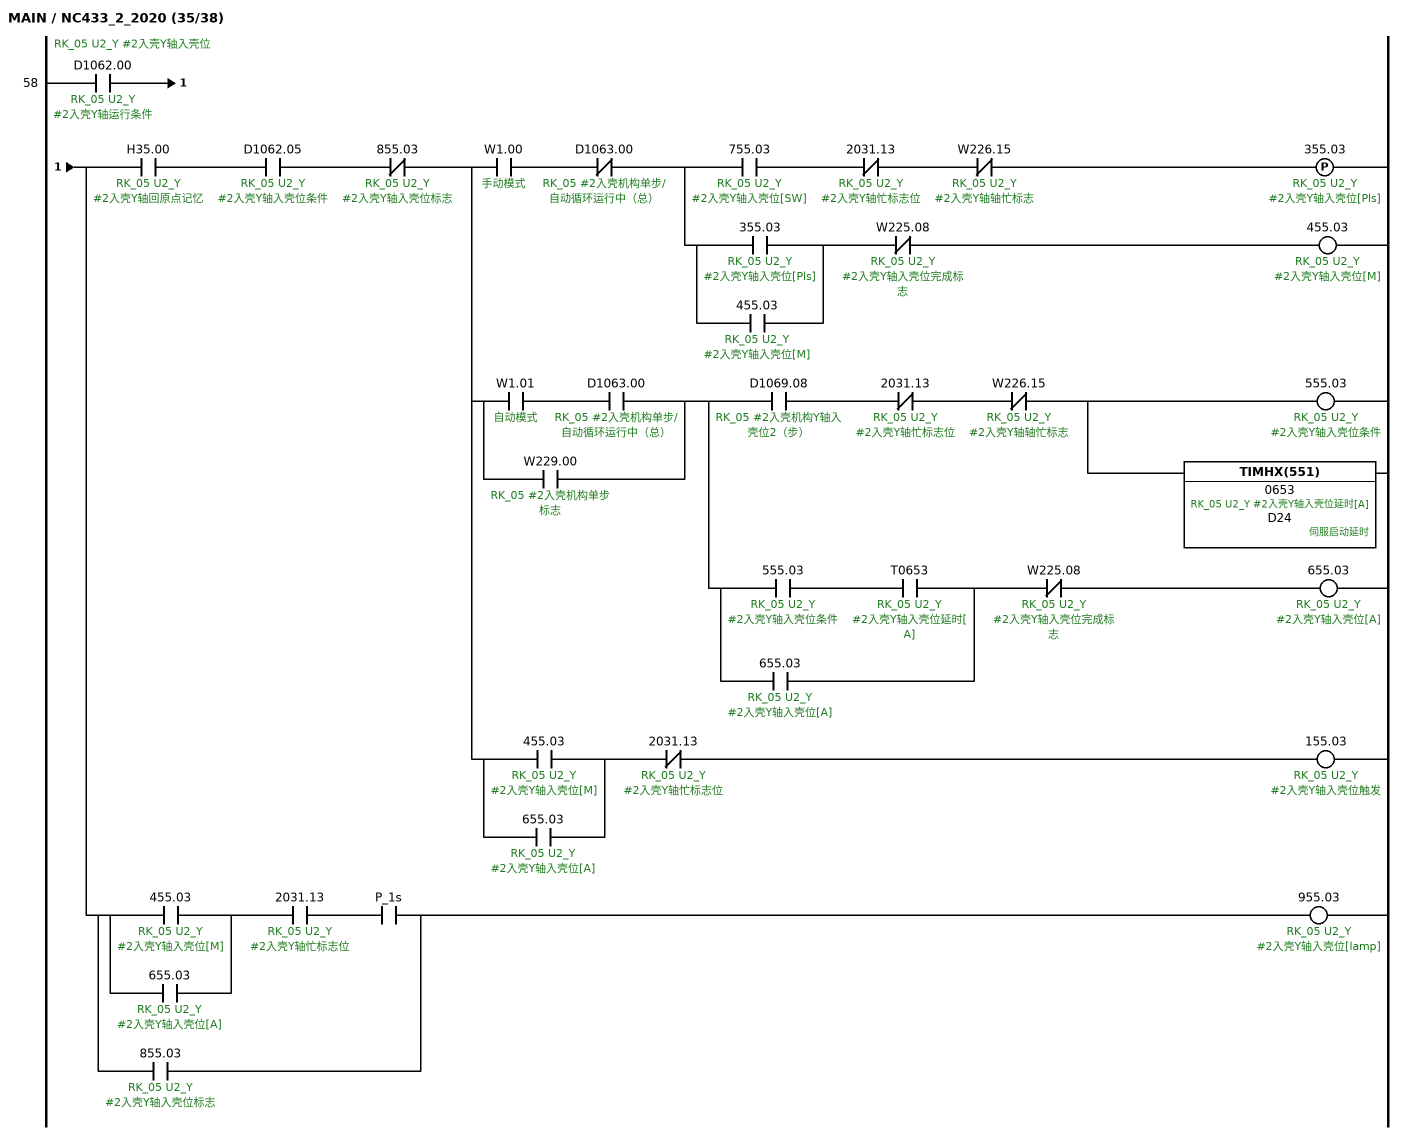
; [picture p144: MAIN / NC433_2_2020, rungs 58-58]
; rung 58: RK_05 U2_Y #2入壳Y轴入壳位
LD D1062.00  ; RK_05 U2_Y #2入壳Y轴运行条件
OUT TR0
AND H35.00  ; RK_05 U2_Y #2入壳Y轴回原点记忆
AND D1062.05  ; RK_05 U2_Y #2入壳Y轴入壳位条件
ANDNOT 855.03  ; RK_05 U2_Y #2入壳Y轴入壳位标志
OUT TR1
AND W1.00  ; 手动模式
ANDNOT D1063.00  ; RK_05 #2入壳机构单步/自动循环运行中（总）
OUT TR2
AND 755.03  ; RK_05 U2_Y #2入壳Y轴入壳位[SW]
ANDNOT 2031.13  ; RK_05 U2_Y #2入壳Y轴忙标志位
ANDNOT W226.15  ; RK_05 U2_Y #2入壳Y轴轴忙标志
DIFU(013) 355.03  ; RK_05 U2_Y #2入壳Y轴入壳位[Pls]
LD TR2
LD 355.03  ; RK_05 U2_Y #2入壳Y轴入壳位[Pls]
OR 455.03  ; RK_05 U2_Y #2入壳Y轴入壳位[M]
ANDLD
ANDNOT W225.08  ; RK_05 U2_Y #2入壳Y轴入壳位完成标志
OUT 455.03  ; RK_05 U2_Y #2入壳Y轴入壳位[M]
LD TR1
LD W1.01  ; 自动模式
AND D1063.00  ; RK_05 #2入壳机构单步/自动循环运行中（总）
OR W229.00  ; RK_05 #2入壳机构单步标志
ANDLD
OUT TR2
AND D1069.08  ; RK_05 #2入壳机构Y轴入壳位2（步）
ANDNOT 2031.13  ; RK_05 U2_Y #2入壳Y轴忙标志位
ANDNOT W226.15  ; RK_05 U2_Y #2入壳Y轴轴忙标志
OUT 555.03  ; RK_05 U2_Y #2入壳Y轴入壳位条件
TIMHX(551) 0653 D24  ; 伺服启动延时, RK_05 U2_Y #2入壳Y轴入壳位延时[A]
LD TR2
LD 555.03  ; RK_05 U2_Y #2入壳Y轴入壳位条件
AND T0653  ; RK_05 U2_Y #2入壳Y轴入壳位延时[A]
OR 655.03  ; RK_05 U2_Y #2入壳Y轴入壳位[A]
ANDLD
ANDNOT W225.08  ; RK_05 U2_Y #2入壳Y轴入壳位完成标志
OUT 655.03  ; RK_05 U2_Y #2入壳Y轴入壳位[A]
LD TR1
LD 455.03  ; RK_05 U2_Y #2入壳Y轴入壳位[M]
OR 655.03  ; RK_05 U2_Y #2入壳Y轴入壳位[A]
ANDLD
ANDNOT 2031.13  ; RK_05 U2_Y #2入壳Y轴忙标志位
OUT 155.03  ; RK_05 U2_Y #2入壳Y轴入壳位触发
LD TR0
LD 455.03  ; RK_05 U2_Y #2入壳Y轴入壳位[M]
OR 655.03  ; RK_05 U2_Y #2入壳Y轴入壳位[A]
AND 2031.13  ; RK_05 U2_Y #2入壳Y轴忙标志位
AND P_1s
OR 855.03  ; RK_05 U2_Y #2入壳Y轴入壳位标志
ANDLD
OUT 955.03  ; RK_05 U2_Y #2入壳Y轴入壳位[lamp]

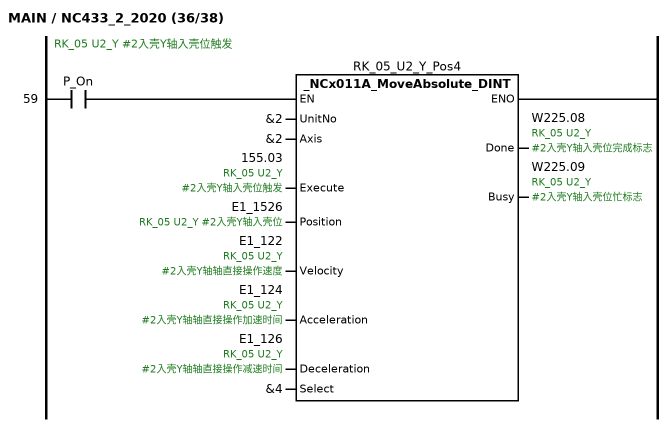
; rung 59: RK_05 U2_Y #2入壳Y轴入壳位触发
LD P_On
CALL RK_05_U2_Y_Pos4 : _NCx011A_MoveAbsolute_DINT (UnitNo := &2, Axis := &2, Execute := 155.03, Position := E1_1526, Velocity := E1_122, Acceleration := E1_124, Deceleration := E1_126, Select := &4, Done => W225.08, Busy => W225.09)  ; RK_05 U2_Y #2入壳Y轴入壳位触发, RK_05 U2_Y #2入壳Y轴入壳位, RK_05 U2_Y #2入壳Y轴轴直接操作速度, RK_05 U2_Y #2入壳Y轴轴直接操作加速时间, RK_05 U2_Y #2入壳Y轴轴直接操作减速时间, RK_05 U2_Y #2入壳Y轴入壳位完成标志, RK_05 U2_Y #2入壳Y轴入壳位忙标志

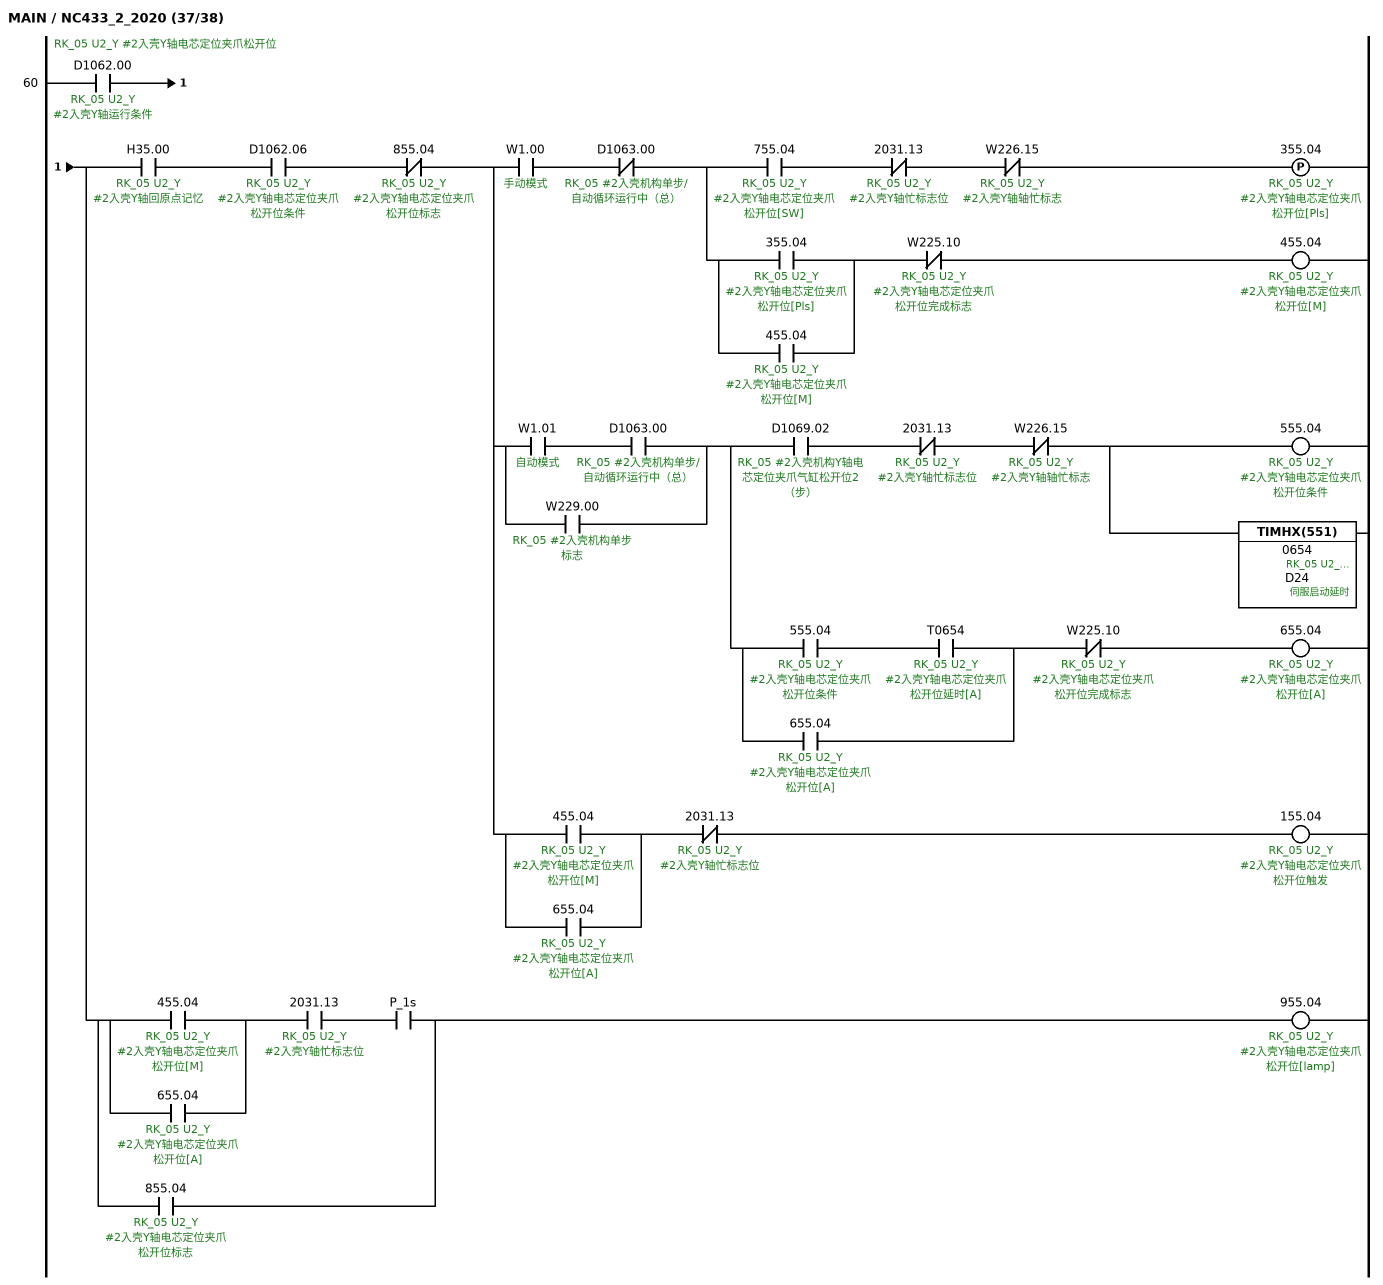
; rung 60: RK_05 U2_Y #2入壳Y轴电芯定位夹爪松开位
LD D1062.00  ; RK_05 U2_Y #2入壳Y轴运行条件
OUT TR0
AND H35.00  ; RK_05 U2_Y #2入壳Y轴回原点记忆
AND D1062.06  ; RK_05 U2_Y #2入壳Y轴电芯定位夹爪松开位条件
ANDNOT 855.04  ; RK_05 U2_Y #2入壳Y轴电芯定位夹爪松开位标志
OUT TR1
AND W1.00  ; 手动模式
ANDNOT D1063.00  ; RK_05 #2入壳机构单步/自动循环运行中（总）
OUT TR2
AND 755.04  ; RK_05 U2_Y #2入壳Y轴电芯定位夹爪松开位[SW]
ANDNOT 2031.13  ; RK_05 U2_Y #2入壳Y轴忙标志位
ANDNOT W226.15  ; RK_05 U2_Y #2入壳Y轴轴忙标志
DIFU(013) 355.04  ; RK_05 U2_Y #2入壳Y轴电芯定位夹爪松开位[Pls]
LD TR2
LD 355.04  ; RK_05 U2_Y #2入壳Y轴电芯定位夹爪松开位[Pls]
OR 455.04  ; RK_05 U2_Y #2入壳Y轴电芯定位夹爪松开位[M]
ANDLD
ANDNOT W225.10  ; RK_05 U2_Y #2入壳Y轴电芯定位夹爪松开位完成标志
OUT 455.04  ; RK_05 U2_Y #2入壳Y轴电芯定位夹爪松开位[M]
LD TR1
LD W1.01  ; 自动模式
AND D1063.00  ; RK_05 #2入壳机构单步/自动循环运行中（总）
OR W229.00  ; RK_05 #2入壳机构单步标志
ANDLD
OUT TR2
AND D1069.02  ; RK_05 #2入壳机构Y轴电芯定位夹爪气缸松开位2（步）
ANDNOT 2031.13  ; RK_05 U2_Y #2入壳Y轴忙标志位
ANDNOT W226.15  ; RK_05 U2_Y #2入壳Y轴轴忙标志
OUT 555.04  ; RK_05 U2_Y #2入壳Y轴电芯定位夹爪松开位条件
TIMHX(551) 0654 D24  ; 伺服启动延时, RK_05 U2_Y #2入壳Y轴电芯定位夹爪松开位延时[A]
LD TR2
LD 555.04  ; RK_05 U2_Y #2入壳Y轴电芯定位夹爪松开位条件
AND T0654  ; RK_05 U2_Y #2入壳Y轴电芯定位夹爪松开位延时[A]
OR 655.04  ; RK_05 U2_Y #2入壳Y轴电芯定位夹爪松开位[A]
ANDLD
ANDNOT W225.10  ; RK_05 U2_Y #2入壳Y轴电芯定位夹爪松开位完成标志
OUT 655.04  ; RK_05 U2_Y #2入壳Y轴电芯定位夹爪松开位[A]
LD TR1
LD 455.04  ; RK_05 U2_Y #2入壳Y轴电芯定位夹爪松开位[M]
OR 655.04  ; RK_05 U2_Y #2入壳Y轴电芯定位夹爪松开位[A]
ANDLD
ANDNOT 2031.13  ; RK_05 U2_Y #2入壳Y轴忙标志位
OUT 155.04  ; RK_05 U2_Y #2入壳Y轴电芯定位夹爪松开位触发
LD TR0
LD 455.04  ; RK_05 U2_Y #2入壳Y轴电芯定位夹爪松开位[M]
OR 655.04  ; RK_05 U2_Y #2入壳Y轴电芯定位夹爪松开位[A]
AND 2031.13  ; RK_05 U2_Y #2入壳Y轴忙标志位
AND P_1s
OR 855.04  ; RK_05 U2_Y #2入壳Y轴电芯定位夹爪松开位标志
ANDLD
OUT 955.04  ; RK_05 U2_Y #2入壳Y轴电芯定位夹爪松开位[lamp]

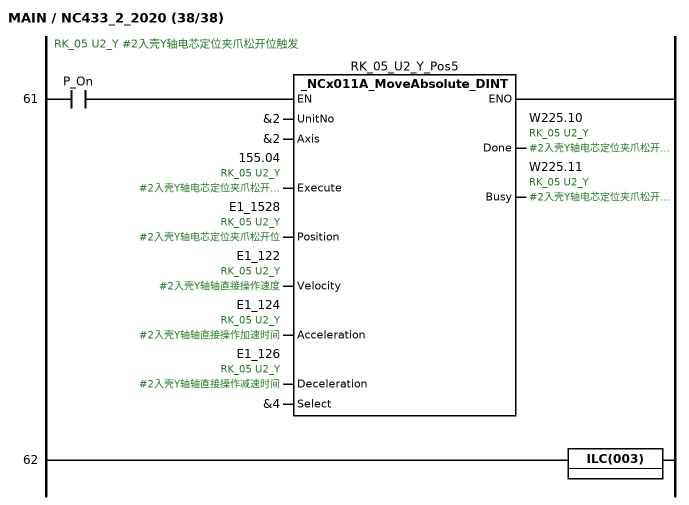
; rung 61: RK_05 U2_Y #2入壳Y轴电芯定位夹爪松开位触发
LD P_On
CALL RK_05_U2_Y_Pos5 : _NCx011A_MoveAbsolute_DINT (UnitNo := &2, Axis := &2, Execute := 155.04, Position := E1_1528, Velocity := E1_122, Acceleration := E1_124, Deceleration := E1_126, Select := &4, Done => W225.10, Busy => W225.11)  ; RK_05 U2_Y #2入壳Y轴电芯定位夹爪松开位触发, RK_05 U2_Y #2入壳Y轴电芯定位夹爪松开位, RK_05 U2_Y #2入壳Y轴轴直接操作速度, RK_05 U2_Y #2入壳Y轴轴直接操作加速时间, RK_05 U2_Y #2入壳Y轴轴直接操作减速时间, RK_05 U2_Y #2入壳Y轴电芯定位夹爪松开位完成标志, RK_05 U2_Y #2入壳Y轴电芯定位夹爪松开位忙标志
; rung 62
ILC(003)

### Section NC433_4_2040

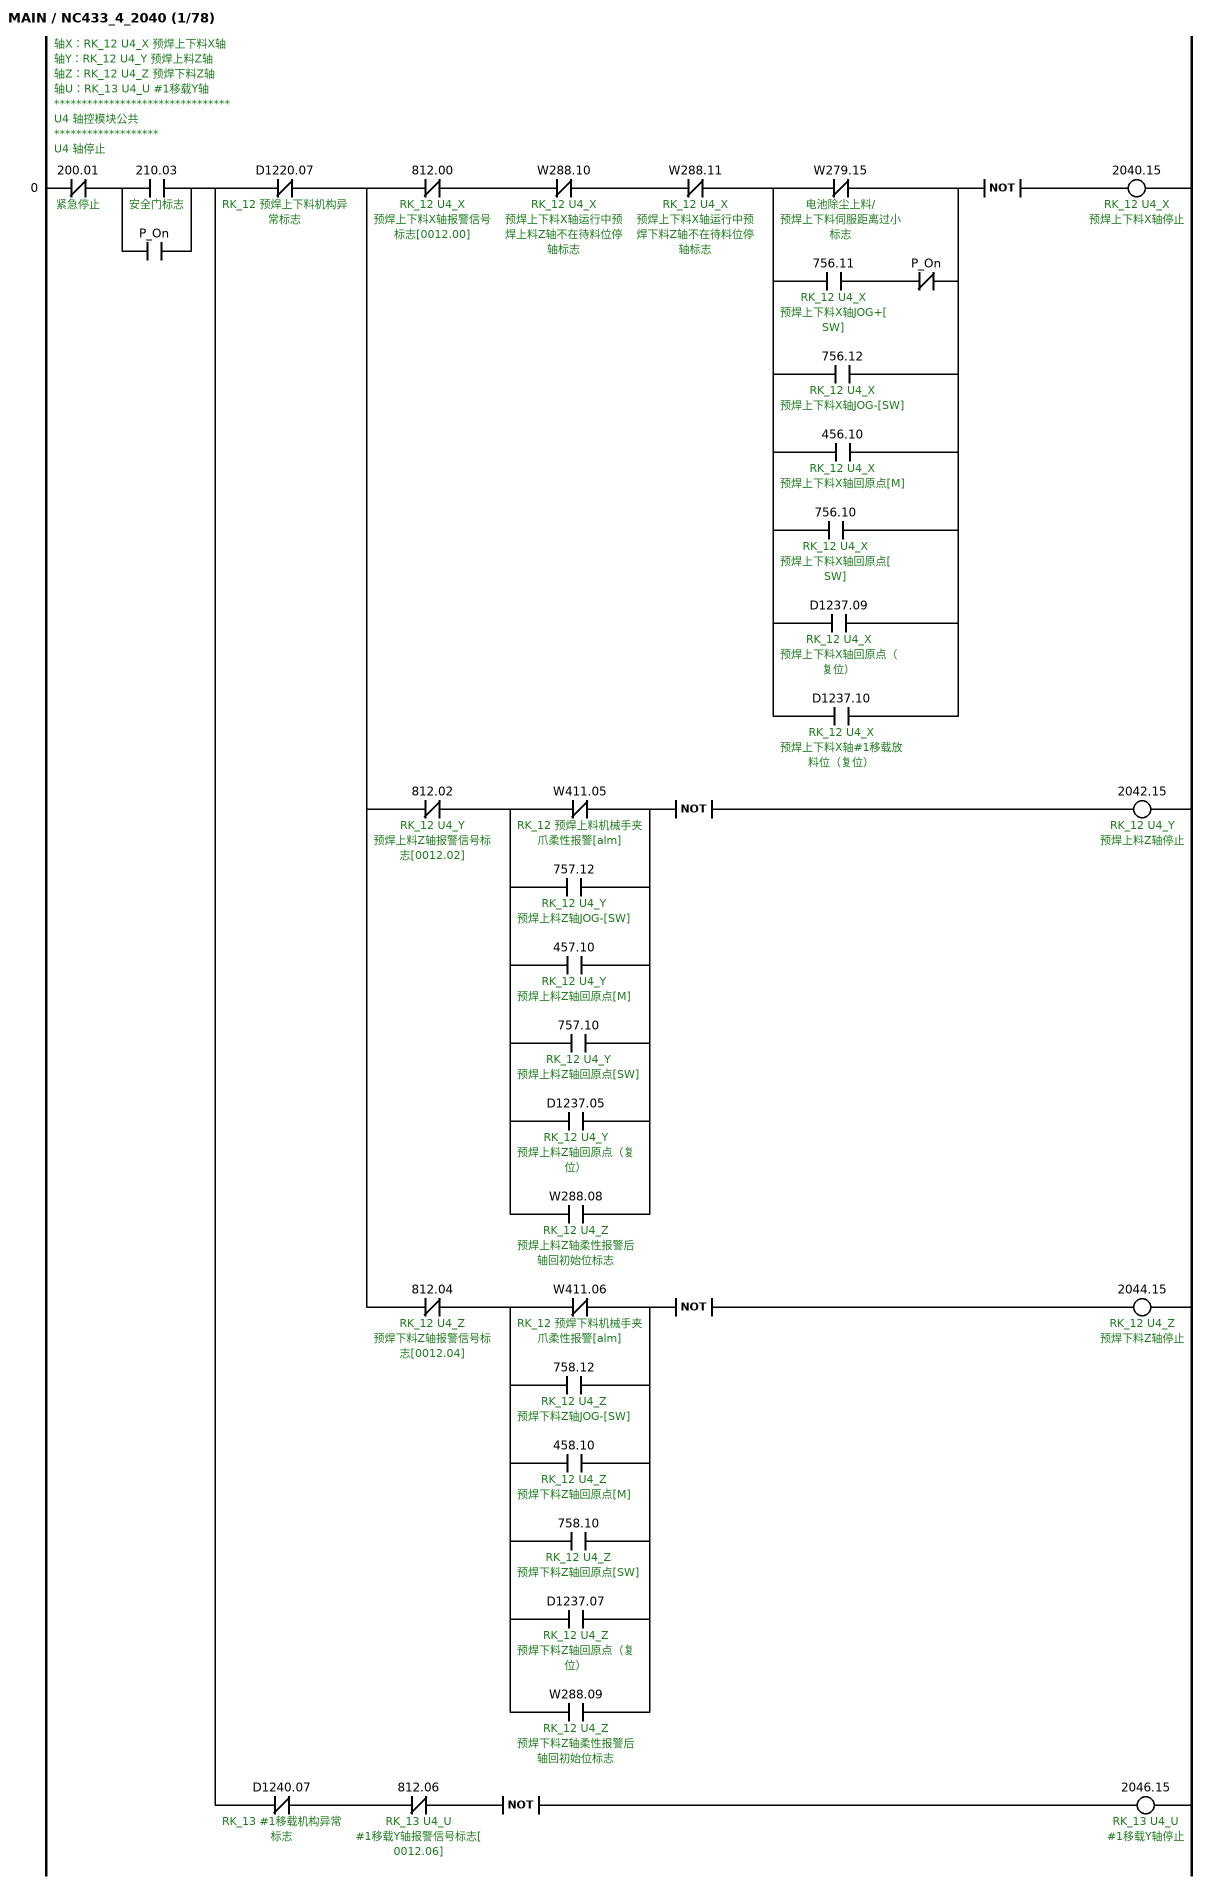
; rung 0: 轴X：RK_12 U4_X 预焊上下料X轴 / 轴Y：RK_12 U4_Y 预焊上料Z轴 / 轴Z：RK_12 U4_Z 预焊下料Z轴 / 轴U：RK_13 U4_U #1移载Y轴 / ******************************** / U4 轴控模块公共 / ******************* / U4 轴停止
LDNOT 200.01  ; 紧急停止
LD 210.03  ; 安全门标志
OR P_On
ANDLD
OUT TR0
ANDNOT D1220.07  ; RK_12 预焊上下料机构异常标志
OUT TR1
ANDNOT 812.00  ; RK_12 U4_X 预焊上下料X轴报警信号标志[0012.00]
ANDNOT W288.10  ; RK_12 U4_X 预焊上下料X轴运行中预焊上料Z轴不在待料位停轴标志
ANDNOT W288.11  ; RK_12 U4_X 预焊上下料X轴运行中预焊下料Z轴不在待料位停轴标志
LDNOT W279.15  ; 电池除尘上料/预焊上下料伺服距离过小标志
LD 756.11  ; RK_12 U4_X 预焊上下料X轴JOG+[SW]
ANDNOT P_On
ORLD
OR 756.12  ; RK_12 U4_X 预焊上下料X轴JOG-[SW]
OR 456.10  ; RK_12 U4_X 预焊上下料X轴回原点[M]
OR 756.10  ; RK_12 U4_X 预焊上下料X轴回原点[SW]
OR D1237.09  ; RK_12 U4_X 预焊上下料X轴回原点（复位）
OR D1237.10  ; RK_12 U4_X 预焊上下料X轴#1移载放料位（复位）
ANDLD
NOT(520)
OUT 2040.15  ; RK_12 U4_X 预焊上下料X轴停止
LD TR1
ANDNOT 812.02  ; RK_12 U4_Y 预焊上料Z轴报警信号标志[0012.02]
LDNOT W411.05  ; RK_12 预焊上料机械手夹爪柔性报警[alm]
OR 757.12  ; RK_12 U4_Y 预焊上料Z轴JOG-[SW]
OR 457.10  ; RK_12 U4_Y 预焊上料Z轴回原点[M]
OR 757.10  ; RK_12 U4_Y 预焊上料Z轴回原点[SW]
OR D1237.05  ; RK_12 U4_Y 预焊上料Z轴回原点（复位）
OR W288.08  ; RK_12 U4_Z 预焊上料Z轴柔性报警后轴回初始位标志
ANDLD
NOT(520)
OUT 2042.15  ; RK_12 U4_Y 预焊上料Z轴停止
LD TR1
ANDNOT 812.04  ; RK_12 U4_Z 预焊下料Z轴报警信号标志[0012.04]
LDNOT W411.06  ; RK_12 预焊下料机械手夹爪柔性报警[alm]
OR 758.12  ; RK_12 U4_Z 预焊下料Z轴JOG-[SW]
OR 458.10  ; RK_12 U4_Z 预焊下料Z轴回原点[M]
OR 758.10  ; RK_12 U4_Z 预焊下料Z轴回原点[SW]
OR D1237.07  ; RK_12 U4_Z 预焊下料Z轴回原点（复位）
OR W288.09  ; RK_12 U4_Z 预焊下料Z轴柔性报警后轴回初始位标志
ANDLD
NOT(520)
OUT 2044.15  ; RK_12 U4_Z 预焊下料Z轴停止
LD TR0
ANDNOT D1240.07  ; RK_13 #1移载机构异常标志
ANDNOT 812.06  ; RK_13 U4_U #1移载Y轴报警信号标志[0012.06]
NOT(520)
OUT 2046.15  ; RK_13 U4_U #1移载Y轴停止

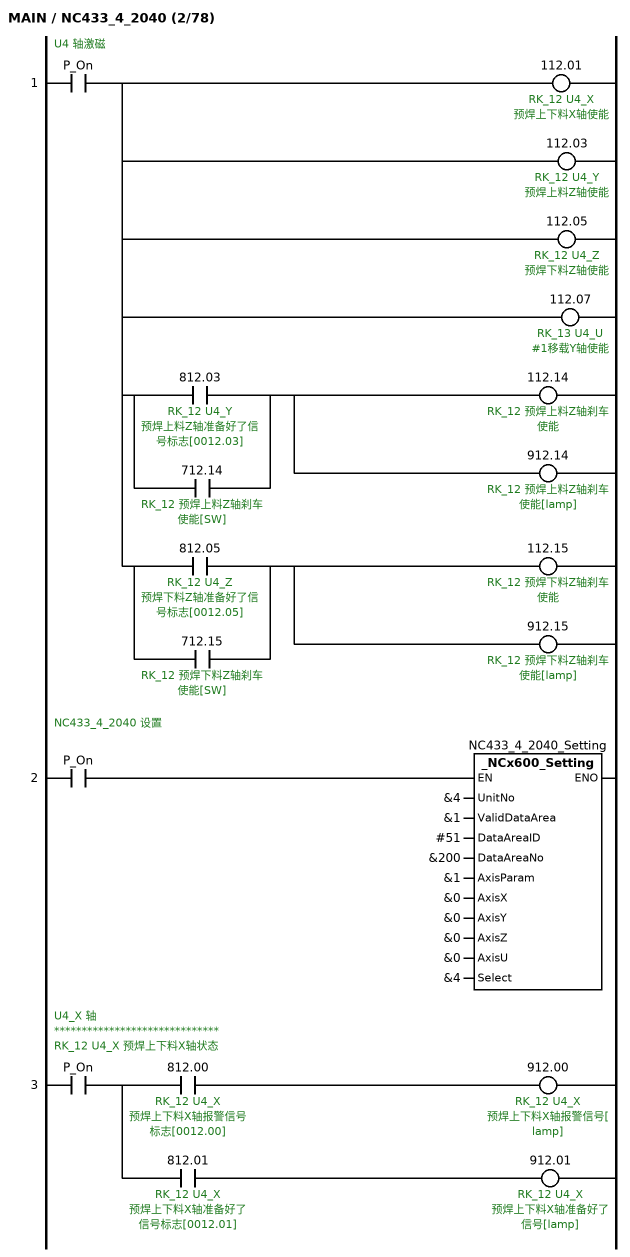
; rung 1: U4 轴激磁
LD P_On
OUT TR0
OUT 112.01  ; RK_12 U4_X 预焊上下料X轴使能
OUT 112.03  ; RK_12 U4_Y 预焊上料Z轴使能
OUT 112.05  ; RK_12 U4_Z 预焊下料Z轴使能
OUT 112.07  ; RK_13 U4_U #1移载Y轴使能
LD 812.03  ; RK_12 U4_Y 预焊上料Z轴准备好了信号标志[0012.03]
OR 712.14  ; RK_12 预焊上料Z轴刹车使能[SW]
ANDLD
OUT 112.14  ; RK_12 预焊上料Z轴刹车使能
OUT 912.14  ; RK_12 预焊上料Z轴刹车使能[lamp]
LD TR0
LD 812.05  ; RK_12 U4_Z 预焊下料Z轴准备好了信号标志[0012.05]
OR 712.15  ; RK_12 预焊下料Z轴刹车使能[SW]
ANDLD
OUT 112.15  ; RK_12 预焊下料Z轴刹车使能
OUT 912.15  ; RK_12 预焊下料Z轴刹车使能[lamp]
; rung 2: NC433_4_2040 设置
LD P_On
CALL NC433_4_2040_Setting : _NCx600_Setting (UnitNo := &4, ValidDataArea := &1, DataAreaID := #51, DataAreaNo := &200, AxisParam := &1, AxisX := &0, AxisY := &0, AxisZ := &0, AxisU := &0, Select := &4)
; rung 3: U4_X 轴 / ****************************** / RK_12 U4_X 预焊上下料X轴状态
LD P_On
OUT TR0
AND 812.00  ; RK_12 U4_X 预焊上下料X轴报警信号标志[0012.00]
OUT 912.00  ; RK_12 U4_X 预焊上下料X轴报警信号[lamp]
LD TR0
AND 812.01  ; RK_12 U4_X 预焊上下料X轴准备好了信号标志[0012.01]
OUT 912.01  ; RK_12 U4_X 预焊上下料X轴准备好了信号[lamp]

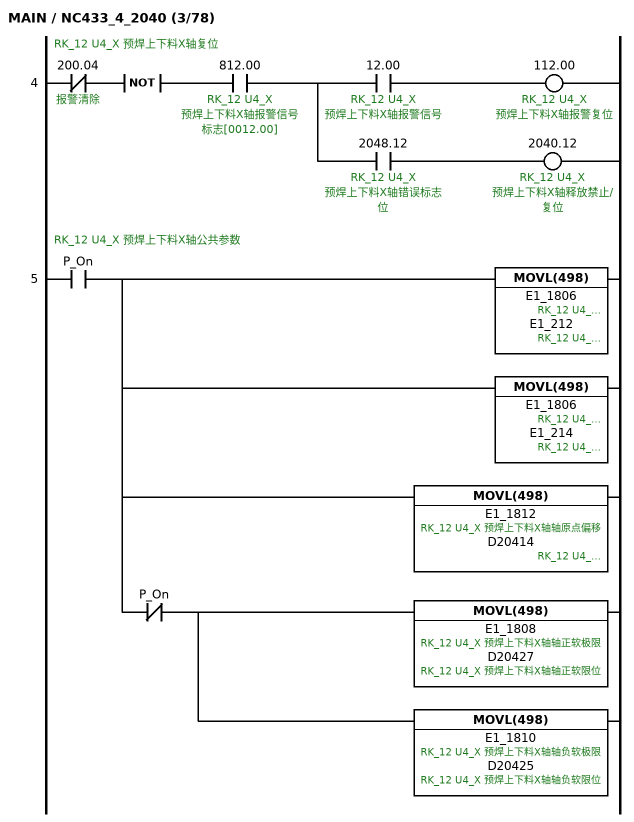
; rung 4: RK_12 U4_X 预焊上下料X轴复位
LDNOT 200.04  ; 报警清除
NOT(520)
AND 812.00  ; RK_12 U4_X 预焊上下料X轴报警信号标志[0012.00]
OUT TR0
AND 12.00  ; RK_12 U4_X 预焊上下料X轴报警信号
OUT 112.00  ; RK_12 U4_X 预焊上下料X轴报警复位
LD TR0
AND 2048.12  ; RK_12 U4_X 预焊上下料X轴错误标志位
OUT 2040.12  ; RK_12 U4_X 预焊上下料X轴释放禁止/复位
; rung 5: RK_12 U4_X 预焊上下料X轴公共参数
LD P_On
MOVL(498) E1_1806 E1_212  ; RK_12 U4_X 预焊上下料X轴轴加减速时间, RK_12 U4_X 预焊上下料X轴轴直接操作加速时间
MOVL(498) E1_1806 E1_214  ; RK_12 U4_X 预焊上下料X轴轴加减速时间, RK_12 U4_X 预焊上下料X轴轴直接操作减速时间
MOVL(498) E1_1812 D20414  ; RK_12 U4_X 预焊上下料X轴轴原点偏移, RK_12 U4_X 预焊上下料X轴轴原点补偿值
ANDNOT P_On
MOVL(498) E1_1808 D20427  ; RK_12 U4_X 预焊上下料X轴轴正软极限, RK_12 U4_X 预焊上下料X轴轴正软限位
MOVL(498) E1_1810 D20425  ; RK_12 U4_X 预焊上下料X轴轴负软极限, RK_12 U4_X 预焊上下料X轴轴负软限位

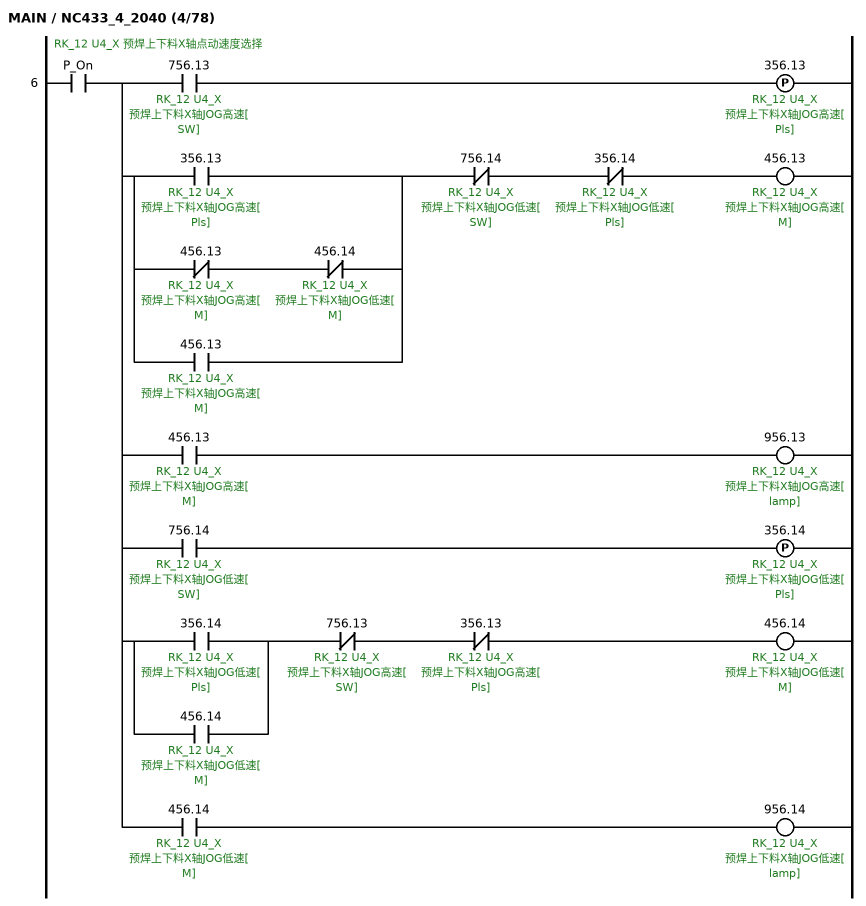
; rung 6: RK_12 U4_X 预焊上下料X轴点动速度选择
LD P_On
OUT TR0
AND 756.13  ; RK_12 U4_X 预焊上下料X轴JOG高速[SW]
DIFU(013) 356.13  ; RK_12 U4_X 预焊上下料X轴JOG高速[Pls]
LD TR0
LD 356.13  ; RK_12 U4_X 预焊上下料X轴JOG高速[Pls]
LDNOT 456.13  ; RK_12 U4_X 预焊上下料X轴JOG高速[M]
ANDNOT 456.14  ; RK_12 U4_X 预焊上下料X轴JOG低速[M]
ORLD
OR 456.13  ; RK_12 U4_X 预焊上下料X轴JOG高速[M]
ANDLD
ANDNOT 756.14  ; RK_12 U4_X 预焊上下料X轴JOG低速[SW]
ANDNOT 356.14  ; RK_12 U4_X 预焊上下料X轴JOG低速[Pls]
OUT 456.13  ; RK_12 U4_X 预焊上下料X轴JOG高速[M]
LD TR0
AND 456.13  ; RK_12 U4_X 预焊上下料X轴JOG高速[M]
OUT 956.13  ; RK_12 U4_X 预焊上下料X轴JOG高速[lamp]
LD TR0
AND 756.14  ; RK_12 U4_X 预焊上下料X轴JOG低速[SW]
DIFU(013) 356.14  ; RK_12 U4_X 预焊上下料X轴JOG低速[Pls]
LD TR0
LD 356.14  ; RK_12 U4_X 预焊上下料X轴JOG低速[Pls]
OR 456.14  ; RK_12 U4_X 预焊上下料X轴JOG低速[M]
ANDLD
ANDNOT 756.13  ; RK_12 U4_X 预焊上下料X轴JOG高速[SW]
ANDNOT 356.13  ; RK_12 U4_X 预焊上下料X轴JOG高速[Pls]
OUT 456.14  ; RK_12 U4_X 预焊上下料X轴JOG低速[M]
LD TR0
AND 456.14  ; RK_12 U4_X 预焊上下料X轴JOG低速[M]
OUT 956.14  ; RK_12 U4_X 预焊上下料X轴JOG低速[lamp]

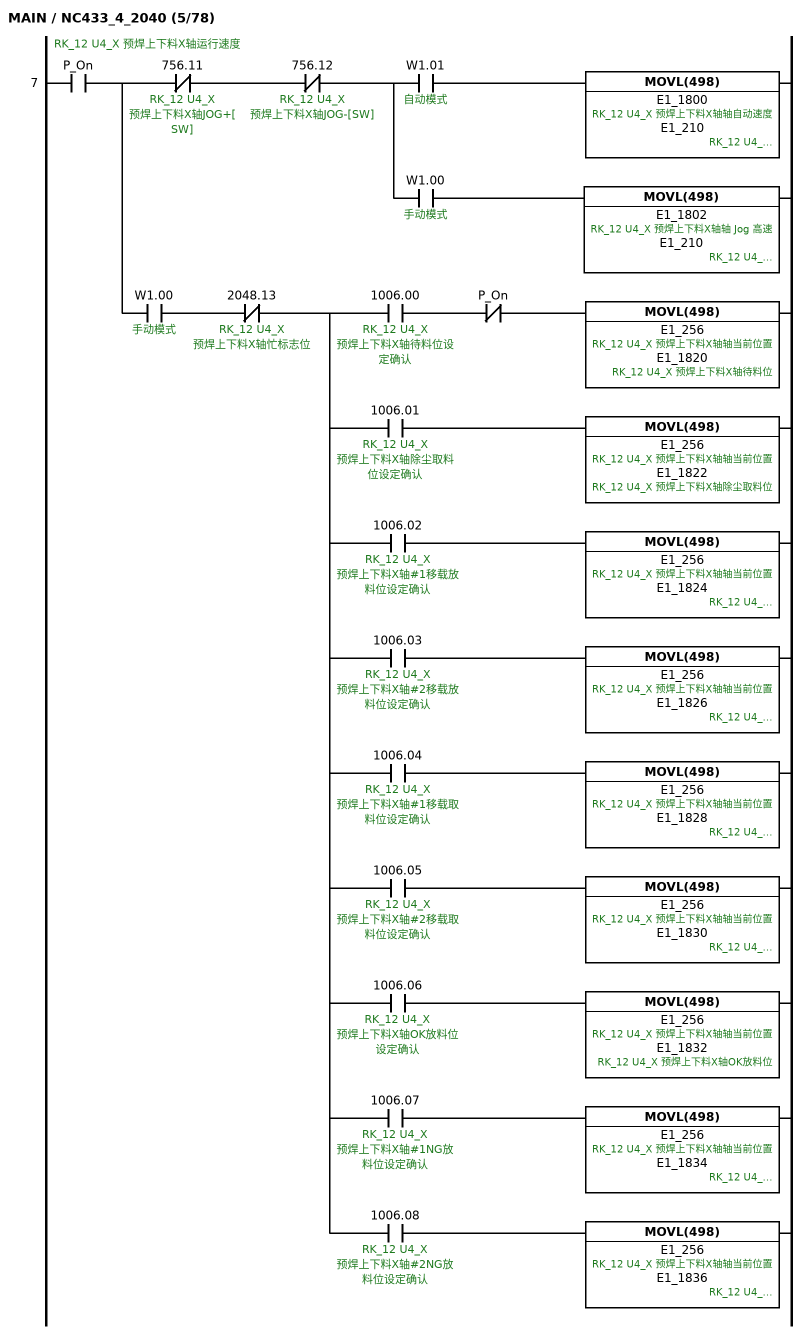
; rung 7: RK_12 U4_X 预焊上下料X轴运行速度
LD P_On
OUT TR0
ANDNOT 756.11  ; RK_12 U4_X 预焊上下料X轴JOG+[SW]
ANDNOT 756.12  ; RK_12 U4_X 预焊上下料X轴JOG-[SW]
OUT TR1
AND W1.01  ; 自动模式
MOVL(498) E1_1800 E1_210  ; RK_12 U4_X 预焊上下料X轴轴自动速度, RK_12 U4_X 预焊上下料X轴轴直接操作速度
LD TR1
AND W1.00  ; 手动模式
MOVL(498) E1_1802 E1_210  ; RK_12 U4_X 预焊上下料X轴轴 Jog 高速, RK_12 U4_X 预焊上下料X轴轴直接操作速度
LD TR0
AND W1.00  ; 手动模式
ANDNOT 2048.13  ; RK_12 U4_X 预焊上下料X轴忙标志位
OUT TR0
AND 1006.00  ; RK_12 U4_X 预焊上下料X轴待料位设定确认
ANDNOT P_On
MOVL(498) E1_256 E1_1820  ; RK_12 U4_X 预焊上下料X轴轴当前位置, RK_12 U4_X 预焊上下料X轴待料位
LD TR0
AND 1006.01  ; RK_12 U4_X 预焊上下料X轴除尘取料位设定确认
MOVL(498) E1_256 E1_1822  ; RK_12 U4_X 预焊上下料X轴轴当前位置, RK_12 U4_X 预焊上下料X轴除尘取料位
LD TR0
AND 1006.02  ; RK_12 U4_X 预焊上下料X轴#1移载放料位设定确认
MOVL(498) E1_256 E1_1824  ; RK_12 U4_X 预焊上下料X轴轴当前位置, RK_12 U4_X 预焊上下料X轴#1移载放料位
LD TR0
AND 1006.03  ; RK_12 U4_X 预焊上下料X轴#2移载放料位设定确认
MOVL(498) E1_256 E1_1826  ; RK_12 U4_X 预焊上下料X轴轴当前位置, RK_12 U4_X 预焊上下料X轴#2移载放料位
LD TR0
AND 1006.04  ; RK_12 U4_X 预焊上下料X轴#1移载取料位设定确认
MOVL(498) E1_256 E1_1828  ; RK_12 U4_X 预焊上下料X轴轴当前位置, RK_12 U4_X 预焊上下料X轴#1移载取料位
LD TR0
AND 1006.05  ; RK_12 U4_X 预焊上下料X轴#2移载取料位设定确认
MOVL(498) E1_256 E1_1830  ; RK_12 U4_X 预焊上下料X轴轴当前位置, RK_12 U4_X 预焊上下料X轴#2移载取料位
LD TR0
AND 1006.06  ; RK_12 U4_X 预焊上下料X轴OK放料位设定确认
MOVL(498) E1_256 E1_1832  ; RK_12 U4_X 预焊上下料X轴轴当前位置, RK_12 U4_X 预焊上下料X轴OK放料位
LD TR0
AND 1006.07  ; RK_12 U4_X 预焊上下料X轴#1NG放料位设定确认
MOVL(498) E1_256 E1_1834  ; RK_12 U4_X 预焊上下料X轴轴当前位置, RK_12 U4_X 预焊上下料X轴#1NG放料位
LD TR0
AND 1006.08  ; RK_12 U4_X 预焊上下料X轴#2NG放料位设定确认
MOVL(498) E1_256 E1_1836  ; RK_12 U4_X 预焊上下料X轴轴当前位置, RK_12 U4_X 预焊上下料X轴#2NG放料位

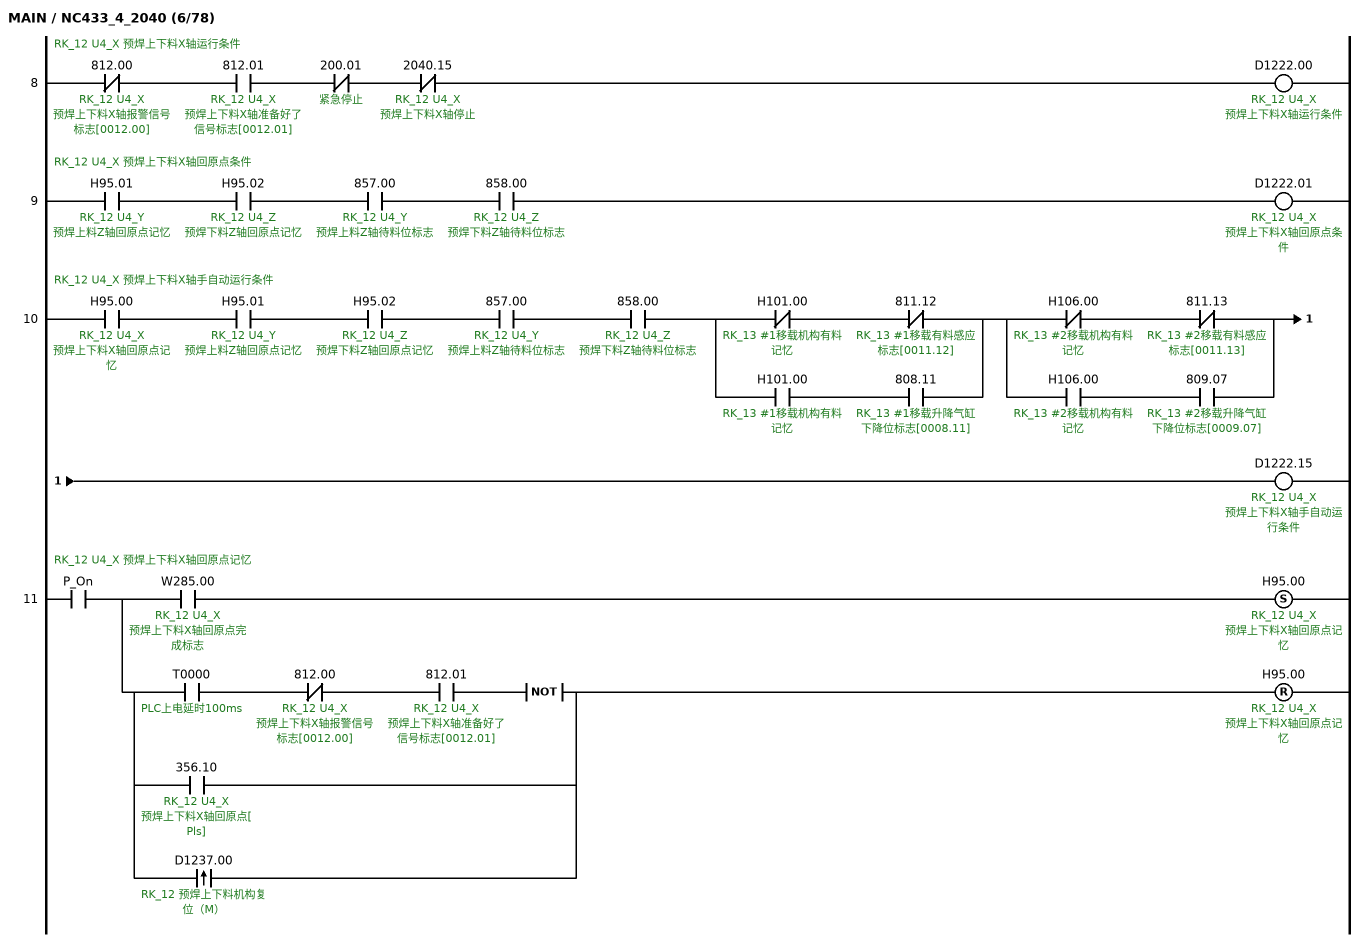
; rung 8: RK_12 U4_X 预焊上下料X轴运行条件
LDNOT 812.00  ; RK_12 U4_X 预焊上下料X轴报警信号标志[0012.00]
AND 812.01  ; RK_12 U4_X 预焊上下料X轴准备好了信号标志[0012.01]
ANDNOT 200.01  ; 紧急停止
ANDNOT 2040.15  ; RK_12 U4_X 预焊上下料X轴停止
OUT D1222.00  ; RK_12 U4_X 预焊上下料X轴运行条件
; rung 9: RK_12 U4_X 预焊上下料X轴回原点条件
LD H95.01  ; RK_12 U4_Y 预焊上料Z轴回原点记忆
AND H95.02  ; RK_12 U4_Z 预焊下料Z轴回原点记忆
AND 857.00  ; RK_12 U4_Y 预焊上料Z轴待料位标志
AND 858.00  ; RK_12 U4_Z 预焊下料Z轴待料位标志
OUT D1222.01  ; RK_12 U4_X 预焊上下料X轴回原点条件
; rung 10: RK_12 U4_X 预焊上下料X轴手自动运行条件
LD H95.00  ; RK_12 U4_X 预焊上下料X轴回原点记忆
AND H95.01  ; RK_12 U4_Y 预焊上料Z轴回原点记忆
AND H95.02  ; RK_12 U4_Z 预焊下料Z轴回原点记忆
AND 857.00  ; RK_12 U4_Y 预焊上料Z轴待料位标志
AND 858.00  ; RK_12 U4_Z 预焊下料Z轴待料位标志
LDNOT H101.00  ; RK_13 #1移载机构有料记忆
ANDNOT 811.12  ; RK_13 #1移载有料感应标志[0011.12]
LD H101.00  ; RK_13 #1移载机构有料记忆
AND 808.11  ; RK_13 #1移载升降气缸下降位标志[0008.11]
ORLD
ANDLD
LDNOT H106.00  ; RK_13 #2移载机构有料记忆
ANDNOT 811.13  ; RK_13 #2移载有料感应标志[0011.13]
LD H106.00  ; RK_13 #2移载机构有料记忆
AND 809.07  ; RK_13 #2移载升降气缸下降位标志[0009.07]
ORLD
ANDLD
OUT D1222.15  ; RK_12 U4_X 预焊上下料X轴手自动运行条件
; rung 11: RK_12 U4_X 预焊上下料X轴回原点记忆
LD P_On
OUT TR0
AND W285.00  ; RK_12 U4_X 预焊上下料X轴回原点完成标志
SET H95.00  ; RK_12 U4_X 预焊上下料X轴回原点记忆
LD TR0
LD T0000  ; PLC上电延时100ms
ANDNOT 812.00  ; RK_12 U4_X 预焊上下料X轴报警信号标志[0012.00]
AND 812.01  ; RK_12 U4_X 预焊上下料X轴准备好了信号标志[0012.01]
NOT(520)
OR 356.10  ; RK_12 U4_X 预焊上下料X轴回原点[Pls]
@OR D1237.00  ; RK_12 预焊上下料机构复位（M）
ANDLD
RSET H95.00  ; RK_12 U4_X 预焊上下料X轴回原点记忆

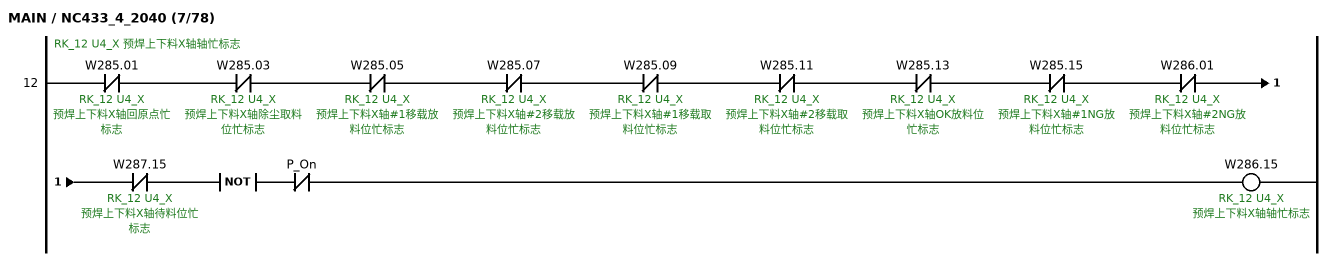
; rung 12: RK_12 U4_X 预焊上下料X轴轴忙标志
LDNOT W285.01  ; RK_12 U4_X 预焊上下料X轴回原点忙标志
ANDNOT W285.03  ; RK_12 U4_X 预焊上下料X轴除尘取料位忙标志
ANDNOT W285.05  ; RK_12 U4_X 预焊上下料X轴#1移载放料位忙标志
ANDNOT W285.07  ; RK_12 U4_X 预焊上下料X轴#2移载放料位忙标志
ANDNOT W285.09  ; RK_12 U4_X 预焊上下料X轴#1移载取料位忙标志
ANDNOT W285.11  ; RK_12 U4_X 预焊上下料X轴#2移载取料位忙标志
ANDNOT W285.13  ; RK_12 U4_X 预焊上下料X轴OK放料位忙标志
ANDNOT W285.15  ; RK_12 U4_X 预焊上下料X轴#1NG放料位忙标志
ANDNOT W286.01  ; RK_12 U4_X 预焊上下料X轴#2NG放料位忙标志
ANDNOT W287.15  ; RK_12 U4_X 预焊上下料X轴待料位忙标志
NOT(520)
ANDNOT P_On
OUT W286.15  ; RK_12 U4_X 预焊上下料X轴轴忙标志

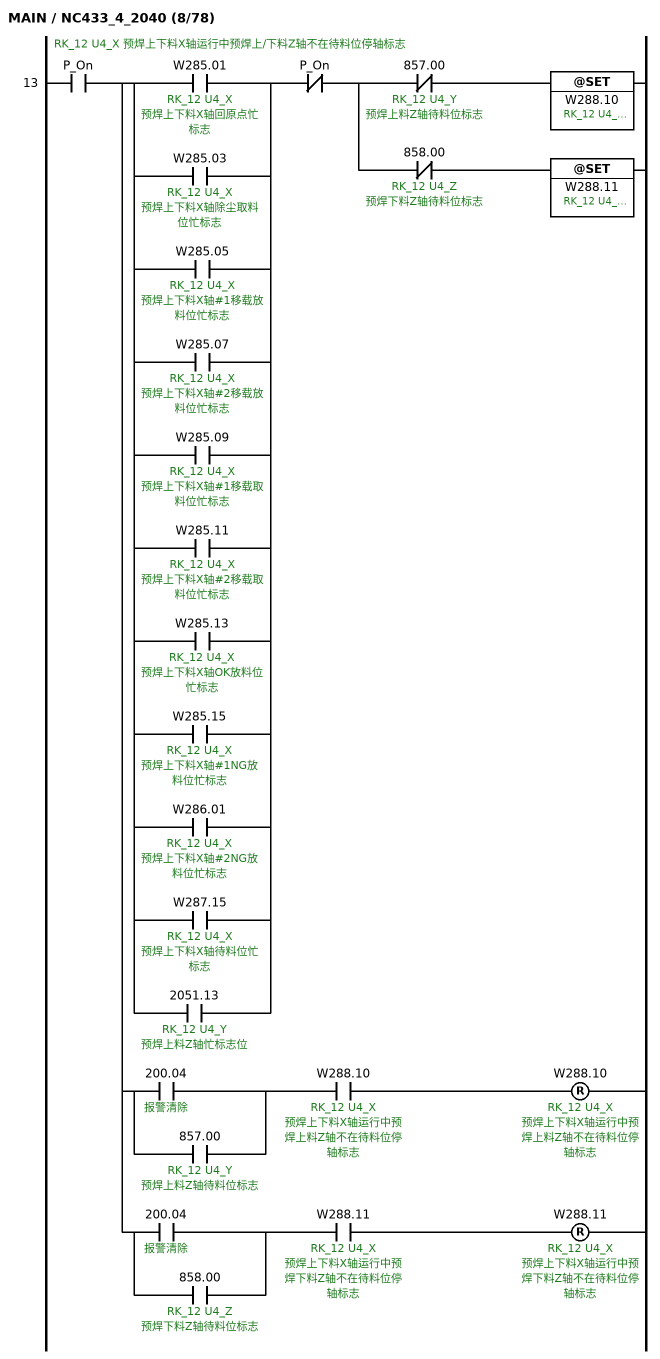
; rung 13: RK_12 U4_X 预焊上下料X轴运行中预焊上/下料Z轴不在待料位停轴标志
LD P_On
OUT TR0
LD W285.01  ; RK_12 U4_X 预焊上下料X轴回原点忙标志
OR W285.03  ; RK_12 U4_X 预焊上下料X轴除尘取料位忙标志
OR W285.05  ; RK_12 U4_X 预焊上下料X轴#1移载放料位忙标志
OR W285.07  ; RK_12 U4_X 预焊上下料X轴#2移载放料位忙标志
OR W285.09  ; RK_12 U4_X 预焊上下料X轴#1移载取料位忙标志
OR W285.11  ; RK_12 U4_X 预焊上下料X轴#2移载取料位忙标志
OR W285.13  ; RK_12 U4_X 预焊上下料X轴OK放料位忙标志
OR W285.15  ; RK_12 U4_X 预焊上下料X轴#1NG放料位忙标志
OR W286.01  ; RK_12 U4_X 预焊上下料X轴#2NG放料位忙标志
OR W287.15  ; RK_12 U4_X 预焊上下料X轴待料位忙标志
OR 2051.13  ; RK_12 U4_Y 预焊上料Z轴忙标志位
ANDLD
ANDNOT P_On
OUT TR1
ANDNOT 857.00  ; RK_12 U4_Y 预焊上料Z轴待料位标志
@SET W288.10  ; RK_12 U4_X 预焊上下料X轴运行中预焊上料Z轴不在待料位停轴标志  // 增加相应报警信息
LD TR1
ANDNOT 858.00  ; RK_12 U4_Z 预焊下料Z轴待料位标志
@SET W288.11  ; RK_12 U4_X 预焊上下料X轴运行中预焊下料Z轴不在待料位停轴标志  // 增加相应报警信息
LD TR0
LD 200.04  ; 报警清除
OR 857.00  ; RK_12 U4_Y 预焊上料Z轴待料位标志
ANDLD
AND W288.10  ; RK_12 U4_X 预焊上下料X轴运行中预焊上料Z轴不在待料位停轴标志
RSET W288.10  ; RK_12 U4_X 预焊上下料X轴运行中预焊上料Z轴不在待料位停轴标志
LD TR0
LD 200.04  ; 报警清除
OR 858.00  ; RK_12 U4_Z 预焊下料Z轴待料位标志
ANDLD
AND W288.11  ; RK_12 U4_X 预焊上下料X轴运行中预焊下料Z轴不在待料位停轴标志
RSET W288.11  ; RK_12 U4_X 预焊上下料X轴运行中预焊下料Z轴不在待料位停轴标志

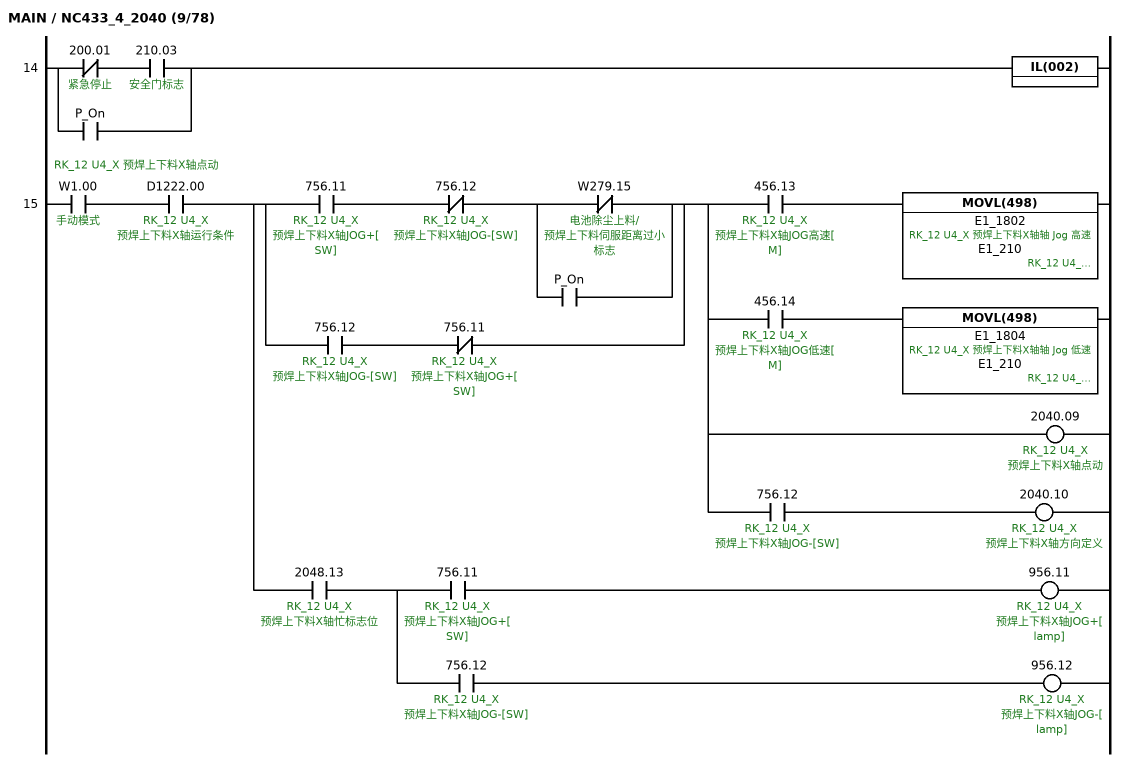
; rung 14
LDNOT 200.01  ; 紧急停止
AND 210.03  ; 安全门标志
OR P_On
IL(002)
; rung 15: RK_12 U4_X 预焊上下料X轴点动
LD W1.00  ; 手动模式
AND D1222.00  ; RK_12 U4_X 预焊上下料X轴运行条件
OUT TR0
LD 756.11  ; RK_12 U4_X 预焊上下料X轴JOG+[SW]
ANDNOT 756.12  ; RK_12 U4_X 预焊上下料X轴JOG-[SW]
LDNOT W279.15  ; 电池除尘上料/预焊上下料伺服距离过小标志
OR P_On
ANDLD
LD 756.12  ; RK_12 U4_X 预焊上下料X轴JOG-[SW]
ANDNOT 756.11  ; RK_12 U4_X 预焊上下料X轴JOG+[SW]
ORLD
ANDLD
OUT TR1
AND 456.13  ; RK_12 U4_X 预焊上下料X轴JOG高速[M]
MOVL(498) E1_1802 E1_210  ; RK_12 U4_X 预焊上下料X轴轴 Jog 高速, RK_12 U4_X 预焊上下料X轴轴直接操作速度
LD TR1
AND 456.14  ; RK_12 U4_X 预焊上下料X轴JOG低速[M]
MOVL(498) E1_1804 E1_210  ; RK_12 U4_X 预焊上下料X轴轴 Jog 低速, RK_12 U4_X 预焊上下料X轴轴直接操作速度
LD TR1
OUT 2040.09  ; RK_12 U4_X 预焊上下料X轴点动
AND 756.12  ; RK_12 U4_X 预焊上下料X轴JOG-[SW]
OUT 2040.10  ; RK_12 U4_X 预焊上下料X轴方向定义
LD TR0
AND 2048.13  ; RK_12 U4_X 预焊上下料X轴忙标志位
OUT TR0
AND 756.11  ; RK_12 U4_X 预焊上下料X轴JOG+[SW]
OUT 956.11  ; RK_12 U4_X 预焊上下料X轴JOG+[lamp]
LD TR0
AND 756.12  ; RK_12 U4_X 预焊上下料X轴JOG-[SW]
OUT 956.12  ; RK_12 U4_X 预焊上下料X轴JOG-[lamp]

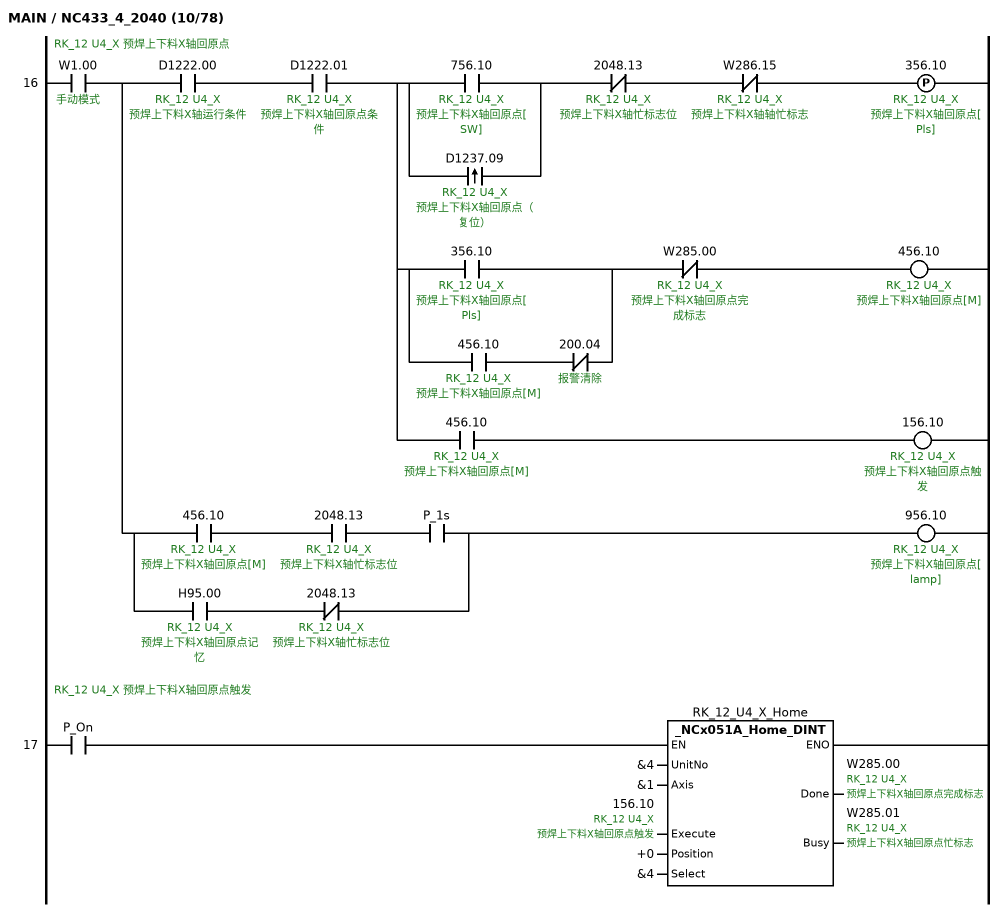
; rung 16: RK_12 U4_X 预焊上下料X轴回原点
LD W1.00  ; 手动模式
OUT TR0
AND D1222.00  ; RK_12 U4_X 预焊上下料X轴运行条件
AND D1222.01  ; RK_12 U4_X 预焊上下料X轴回原点条件
OUT TR1
LD 756.10  ; RK_12 U4_X 预焊上下料X轴回原点[SW]
@OR D1237.09  ; RK_12 U4_X 预焊上下料X轴回原点（复位）
ANDLD
ANDNOT 2048.13  ; RK_12 U4_X 预焊上下料X轴忙标志位
ANDNOT W286.15  ; RK_12 U4_X 预焊上下料X轴轴忙标志
DIFU(013) 356.10  ; RK_12 U4_X 预焊上下料X轴回原点[Pls]
LD TR1
LD 356.10  ; RK_12 U4_X 预焊上下料X轴回原点[Pls]
LD 456.10  ; RK_12 U4_X 预焊上下料X轴回原点[M]
ANDNOT 200.04  ; 报警清除
ORLD
ANDLD
ANDNOT W285.00  ; RK_12 U4_X 预焊上下料X轴回原点完成标志
OUT 456.10  ; RK_12 U4_X 预焊上下料X轴回原点[M]
LD TR1
AND 456.10  ; RK_12 U4_X 预焊上下料X轴回原点[M]
OUT 156.10  ; RK_12 U4_X 预焊上下料X轴回原点触发
LD TR0
LD 456.10  ; RK_12 U4_X 预焊上下料X轴回原点[M]
AND 2048.13  ; RK_12 U4_X 预焊上下料X轴忙标志位
AND P_1s
LD H95.00  ; RK_12 U4_X 预焊上下料X轴回原点记忆
ANDNOT 2048.13  ; RK_12 U4_X 预焊上下料X轴忙标志位
ORLD
ANDLD
OUT 956.10  ; RK_12 U4_X 预焊上下料X轴回原点[lamp]
; rung 17: RK_12 U4_X 预焊上下料X轴回原点触发
LD P_On
CALL RK_12_U4_X_Home : _NCx051A_Home_DINT (UnitNo := &4, Axis := &1, Execute := 156.10, Position := +0, Select := &4, Done => W285.00, Busy => W285.01)  ; RK_12 U4_X 预焊上下料X轴回原点触发, RK_12 U4_X 预焊上下料X轴回原点完成标志, RK_12 U4_X 预焊上下料X轴回原点忙标志

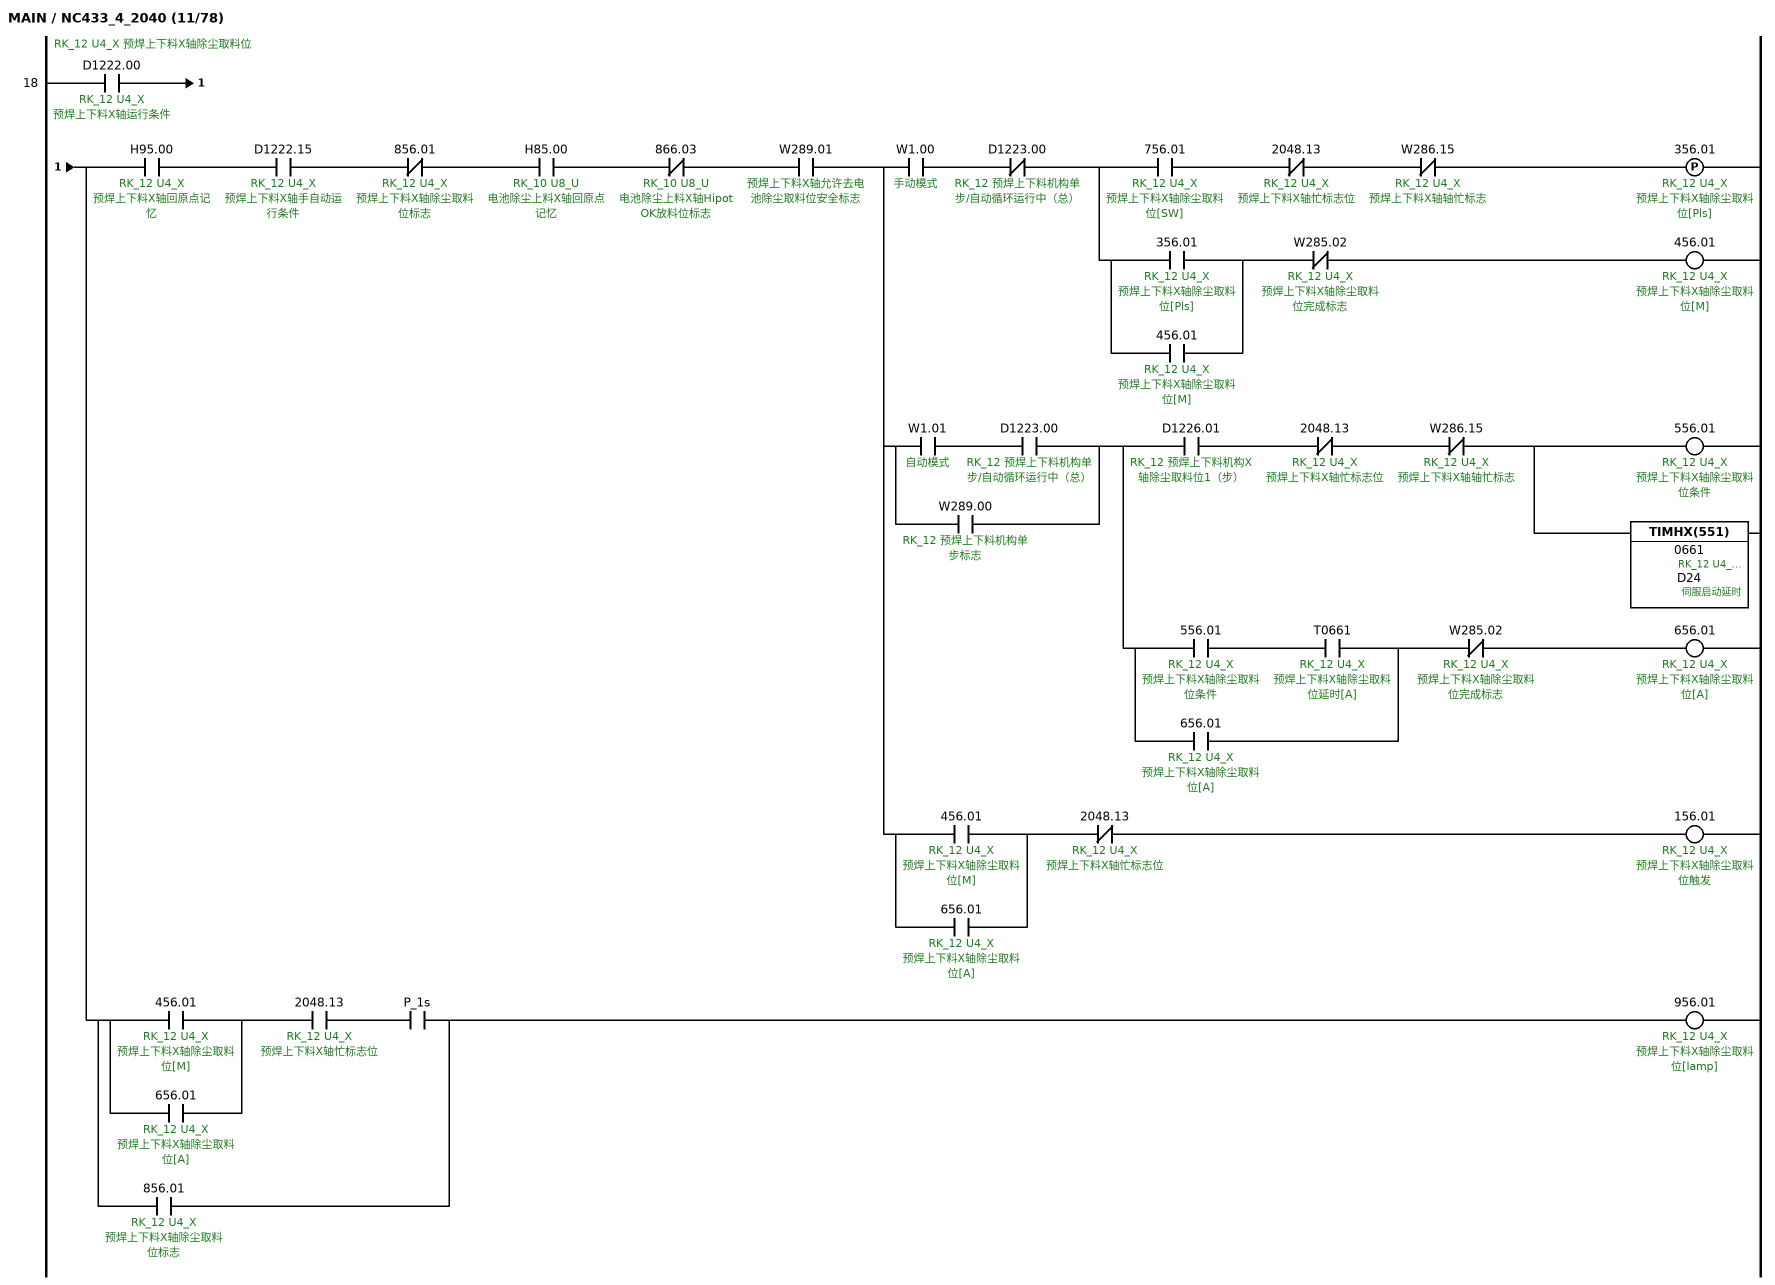
; rung 18: RK_12 U4_X 预焊上下料X轴除尘取料位
LD D1222.00  ; RK_12 U4_X 预焊上下料X轴运行条件
OUT TR0
AND H95.00  ; RK_12 U4_X 预焊上下料X轴回原点记忆
AND D1222.15  ; RK_12 U4_X 预焊上下料X轴手自动运行条件
ANDNOT 856.01  ; RK_12 U4_X 预焊上下料X轴除尘取料位标志
AND H85.00  ; RK_10 U8_U 电池除尘上料X轴回原点记忆
ANDNOT 866.03  ; RK_10 U8_U 电池除尘上料X轴Hipot OK放料位标志
AND W289.01  ; 预焊上下料X轴允许去电池除尘取料位安全标志
OUT TR1
AND W1.00  ; 手动模式
ANDNOT D1223.00  ; RK_12 预焊上下料机构单步/自动循环运行中（总）
OUT TR2
AND 756.01  ; RK_12 U4_X 预焊上下料X轴除尘取料位[SW]
ANDNOT 2048.13  ; RK_12 U4_X 预焊上下料X轴忙标志位
ANDNOT W286.15  ; RK_12 U4_X 预焊上下料X轴轴忙标志
DIFU(013) 356.01  ; RK_12 U4_X 预焊上下料X轴除尘取料位[Pls]
LD TR2
LD 356.01  ; RK_12 U4_X 预焊上下料X轴除尘取料位[Pls]
OR 456.01  ; RK_12 U4_X 预焊上下料X轴除尘取料位[M]
ANDLD
ANDNOT W285.02  ; RK_12 U4_X 预焊上下料X轴除尘取料位完成标志
OUT 456.01  ; RK_12 U4_X 预焊上下料X轴除尘取料位[M]
LD TR1
LD W1.01  ; 自动模式
AND D1223.00  ; RK_12 预焊上下料机构单步/自动循环运行中（总）
OR W289.00  ; RK_12 预焊上下料机构单步标志
ANDLD
OUT TR2
AND D1226.01  ; RK_12 预焊上下料机构X轴除尘取料位1（步）
ANDNOT 2048.13  ; RK_12 U4_X 预焊上下料X轴忙标志位
ANDNOT W286.15  ; RK_12 U4_X 预焊上下料X轴轴忙标志
OUT 556.01  ; RK_12 U4_X 预焊上下料X轴除尘取料位条件
TIMHX(551) 0661 D24  ; 伺服启动延时, RK_12 U4_X 预焊上下料X轴除尘取料位延时[A]
LD TR2
LD 556.01  ; RK_12 U4_X 预焊上下料X轴除尘取料位条件
AND T0661  ; RK_12 U4_X 预焊上下料X轴除尘取料位延时[A]
OR 656.01  ; RK_12 U4_X 预焊上下料X轴除尘取料位[A]
ANDLD
ANDNOT W285.02  ; RK_12 U4_X 预焊上下料X轴除尘取料位完成标志
OUT 656.01  ; RK_12 U4_X 预焊上下料X轴除尘取料位[A]
LD TR1
LD 456.01  ; RK_12 U4_X 预焊上下料X轴除尘取料位[M]
OR 656.01  ; RK_12 U4_X 预焊上下料X轴除尘取料位[A]
ANDLD
ANDNOT 2048.13  ; RK_12 U4_X 预焊上下料X轴忙标志位
OUT 156.01  ; RK_12 U4_X 预焊上下料X轴除尘取料位触发
LD TR0
LD 456.01  ; RK_12 U4_X 预焊上下料X轴除尘取料位[M]
OR 656.01  ; RK_12 U4_X 预焊上下料X轴除尘取料位[A]
AND 2048.13  ; RK_12 U4_X 预焊上下料X轴忙标志位
AND P_1s
OR 856.01  ; RK_12 U4_X 预焊上下料X轴除尘取料位标志
ANDLD
OUT 956.01  ; RK_12 U4_X 预焊上下料X轴除尘取料位[lamp]

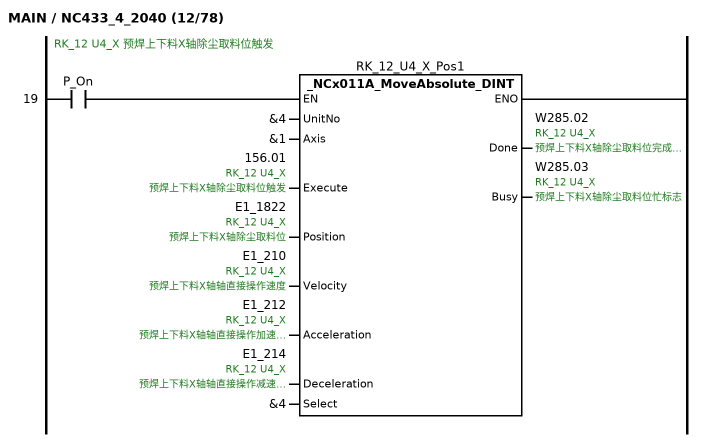
; rung 19: RK_12 U4_X 预焊上下料X轴除尘取料位触发
LD P_On
CALL RK_12_U4_X_Pos1 : _NCx011A_MoveAbsolute_DINT (UnitNo := &4, Axis := &1, Execute := 156.01, Position := E1_1822, Velocity := E1_210, Acceleration := E1_212, Deceleration := E1_214, Select := &4, Done => W285.02, Busy => W285.03)  ; RK_12 U4_X 预焊上下料X轴除尘取料位触发, RK_12 U4_X 预焊上下料X轴除尘取料位, RK_12 U4_X 预焊上下料X轴轴直接操作速度, RK_12 U4_X 预焊上下料X轴轴直接操作加速时间, RK_12 U4_X 预焊上下料X轴轴直接操作减速时间, RK_12 U4_X 预焊上下料X轴除尘取料位完成标志, RK_12 U4_X 预焊上下料X轴除尘取料位忙标志

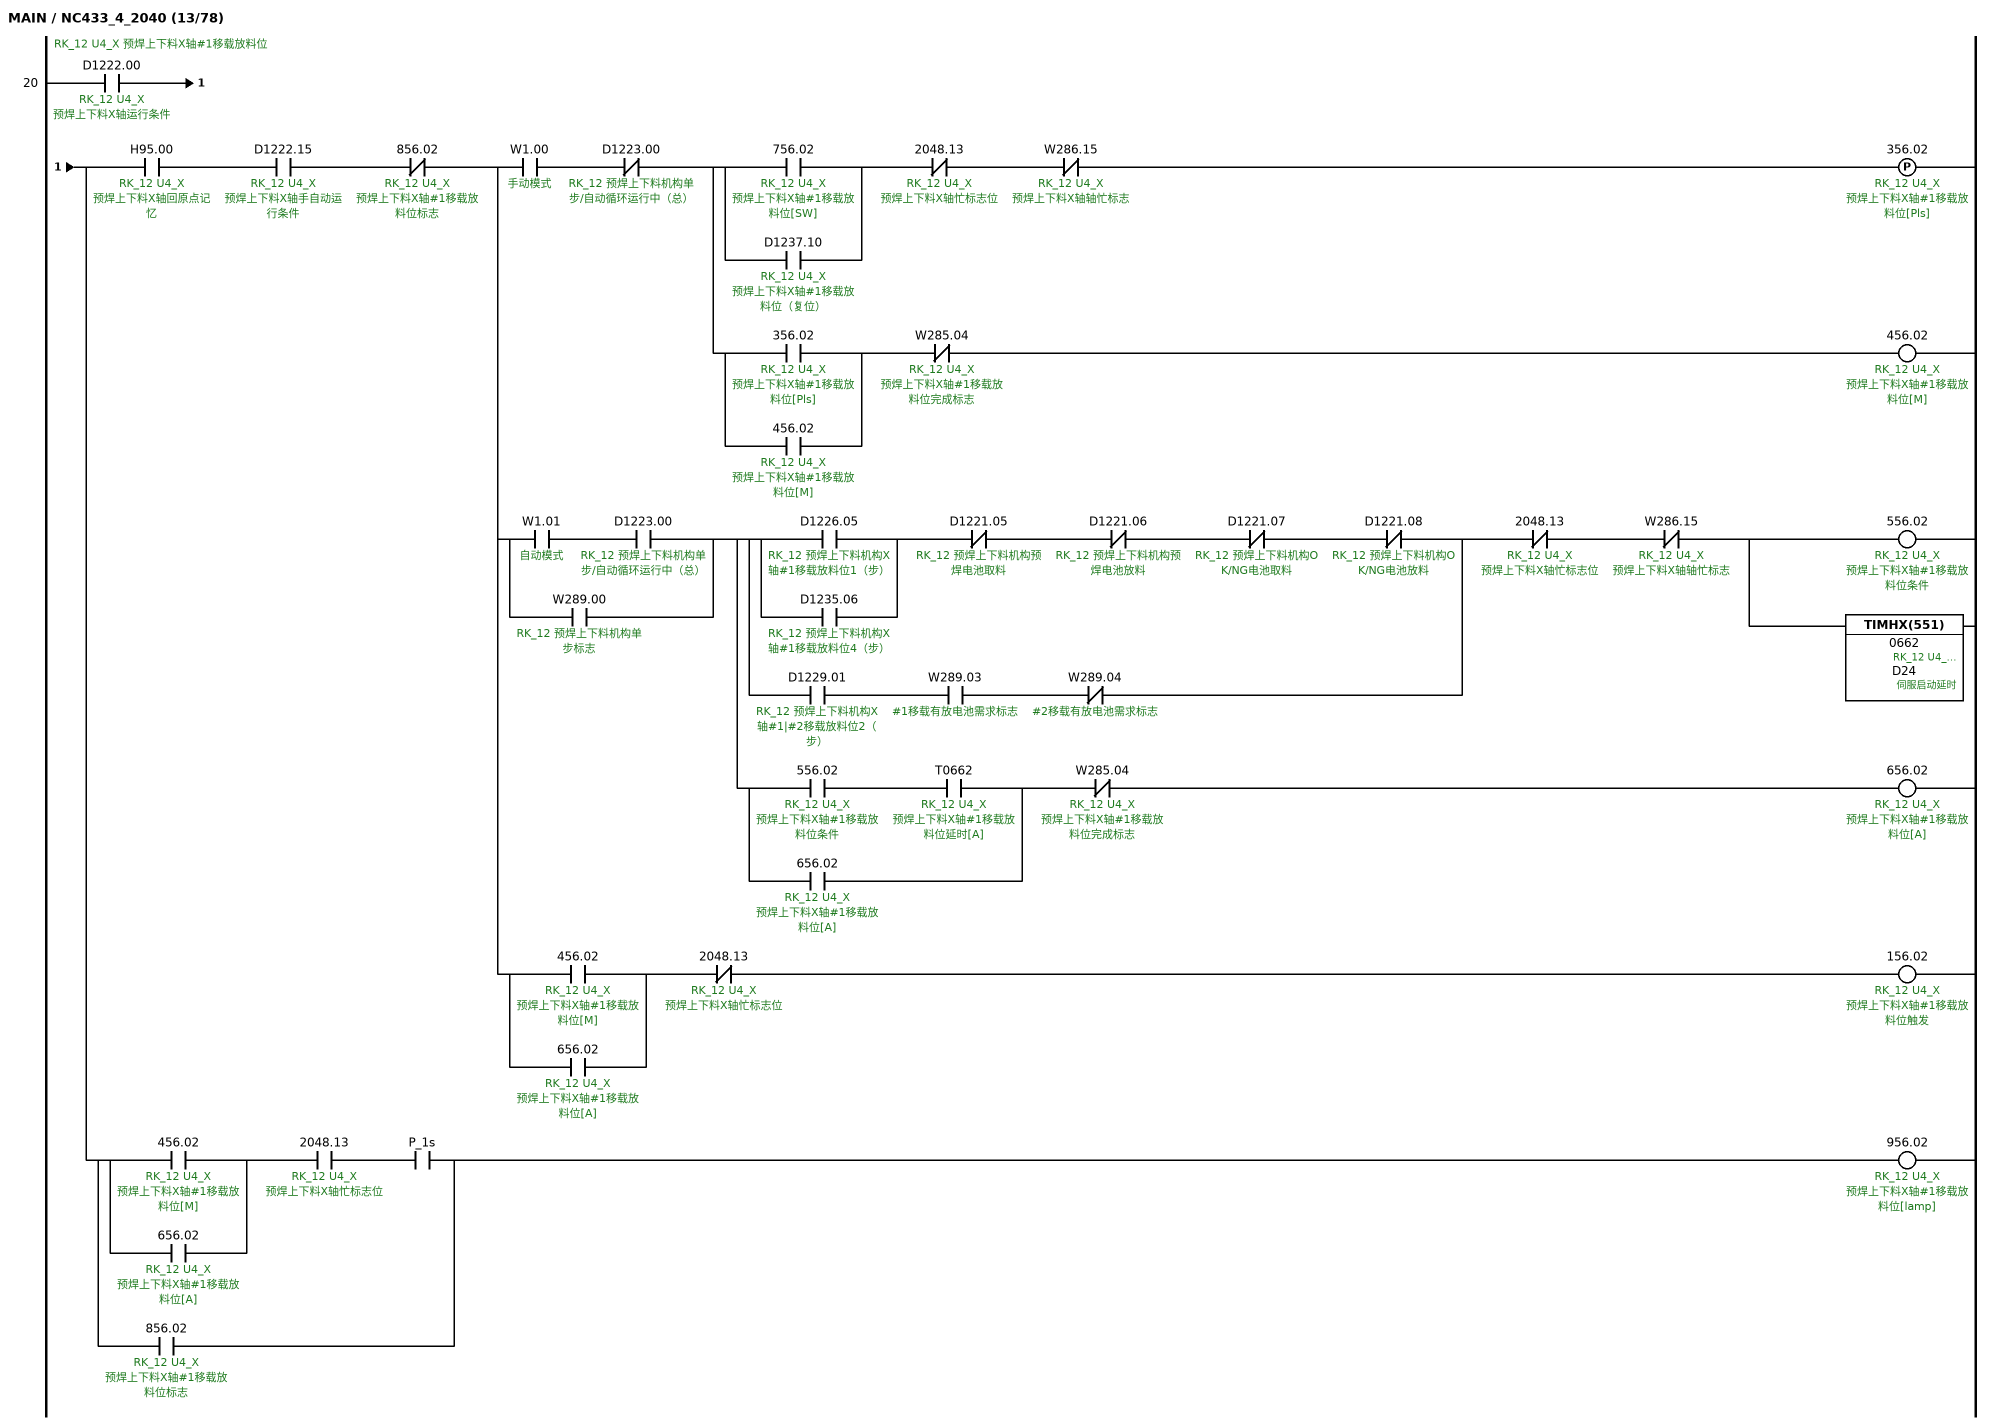
; rung 20: RK_12 U4_X 预焊上下料X轴#1移载放料位
LD D1222.00  ; RK_12 U4_X 预焊上下料X轴运行条件
OUT TR0
AND H95.00  ; RK_12 U4_X 预焊上下料X轴回原点记忆
AND D1222.15  ; RK_12 U4_X 预焊上下料X轴手自动运行条件
ANDNOT 856.02  ; RK_12 U4_X 预焊上下料X轴#1移载放料位标志
OUT TR1
AND W1.00  ; 手动模式
ANDNOT D1223.00  ; RK_12 预焊上下料机构单步/自动循环运行中（总）
OUT TR2
LD 756.02  ; RK_12 U4_X 预焊上下料X轴#1移载放料位[SW]
OR D1237.10  ; RK_12 U4_X 预焊上下料X轴#1移载放料位（复位）
ANDLD
ANDNOT 2048.13  ; RK_12 U4_X 预焊上下料X轴忙标志位
ANDNOT W286.15  ; RK_12 U4_X 预焊上下料X轴轴忙标志
DIFU(013) 356.02  ; RK_12 U4_X 预焊上下料X轴#1移载放料位[Pls]
LD TR2
LD 356.02  ; RK_12 U4_X 预焊上下料X轴#1移载放料位[Pls]
OR 456.02  ; RK_12 U4_X 预焊上下料X轴#1移载放料位[M]
ANDLD
ANDNOT W285.04  ; RK_12 U4_X 预焊上下料X轴#1移载放料位完成标志
OUT 456.02  ; RK_12 U4_X 预焊上下料X轴#1移载放料位[M]
LD TR1
LD W1.01  ; 自动模式
AND D1223.00  ; RK_12 预焊上下料机构单步/自动循环运行中（总）
OR W289.00  ; RK_12 预焊上下料机构单步标志
ANDLD
OUT TR2
LD D1226.05  ; RK_12 预焊上下料机构X轴#1移载放料位1（步）
OR D1235.06  ; RK_12 预焊上下料机构X轴#1移载放料位4（步）
ANDNOT D1221.05  ; RK_12 预焊上下料机构预焊电池取料
ANDNOT D1221.06  ; RK_12 预焊上下料机构预焊电池放料
ANDNOT D1221.07  ; RK_12 预焊上下料机构OK/NG电池取料
ANDNOT D1221.08  ; RK_12 预焊上下料机构OK/NG电池放料
LD D1229.01  ; RK_12 预焊上下料机构X轴#1|#2移载放料位2（步）
AND W289.03  ; #1移载有放电池需求标志
ANDNOT W289.04  ; #2移载有放电池需求标志
ORLD
ANDLD
ANDNOT 2048.13  ; RK_12 U4_X 预焊上下料X轴忙标志位
ANDNOT W286.15  ; RK_12 U4_X 预焊上下料X轴轴忙标志
OUT 556.02  ; RK_12 U4_X 预焊上下料X轴#1移载放料位条件
TIMHX(551) 0662 D24  ; 伺服启动延时, RK_12 U4_X 预焊上下料X轴#1移载放料位延时[A]
LD TR2
LD 556.02  ; RK_12 U4_X 预焊上下料X轴#1移载放料位条件
AND T0662  ; RK_12 U4_X 预焊上下料X轴#1移载放料位延时[A]
OR 656.02  ; RK_12 U4_X 预焊上下料X轴#1移载放料位[A]
ANDLD
ANDNOT W285.04  ; RK_12 U4_X 预焊上下料X轴#1移载放料位完成标志
OUT 656.02  ; RK_12 U4_X 预焊上下料X轴#1移载放料位[A]
LD TR1
LD 456.02  ; RK_12 U4_X 预焊上下料X轴#1移载放料位[M]
OR 656.02  ; RK_12 U4_X 预焊上下料X轴#1移载放料位[A]
ANDLD
ANDNOT 2048.13  ; RK_12 U4_X 预焊上下料X轴忙标志位
OUT 156.02  ; RK_12 U4_X 预焊上下料X轴#1移载放料位触发
LD TR0
LD 456.02  ; RK_12 U4_X 预焊上下料X轴#1移载放料位[M]
OR 656.02  ; RK_12 U4_X 预焊上下料X轴#1移载放料位[A]
AND 2048.13  ; RK_12 U4_X 预焊上下料X轴忙标志位
AND P_1s
OR 856.02  ; RK_12 U4_X 预焊上下料X轴#1移载放料位标志
ANDLD
OUT 956.02  ; RK_12 U4_X 预焊上下料X轴#1移载放料位[lamp]

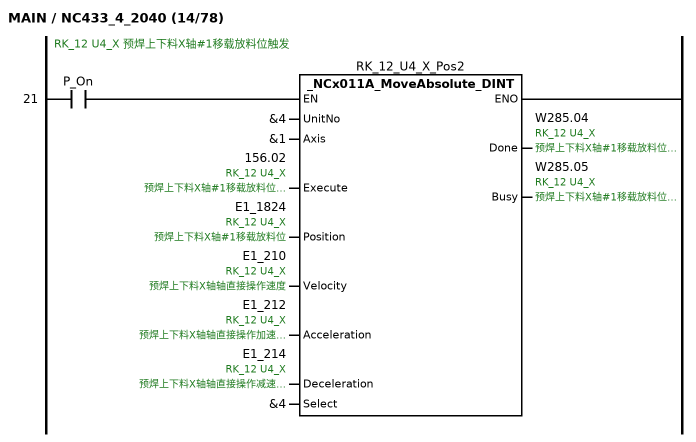
; rung 21: RK_12 U4_X 预焊上下料X轴#1移载放料位触发
LD P_On
CALL RK_12_U4_X_Pos2 : _NCx011A_MoveAbsolute_DINT (UnitNo := &4, Axis := &1, Execute := 156.02, Position := E1_1824, Velocity := E1_210, Acceleration := E1_212, Deceleration := E1_214, Select := &4, Done => W285.04, Busy => W285.05)  ; RK_12 U4_X 预焊上下料X轴#1移载放料位触发, RK_12 U4_X 预焊上下料X轴#1移载放料位, RK_12 U4_X 预焊上下料X轴轴直接操作速度, RK_12 U4_X 预焊上下料X轴轴直接操作加速时间, RK_12 U4_X 预焊上下料X轴轴直接操作减速时间, RK_12 U4_X 预焊上下料X轴#1移载放料位完成标志, RK_12 U4_X 预焊上下料X轴#1移载放料位忙标志

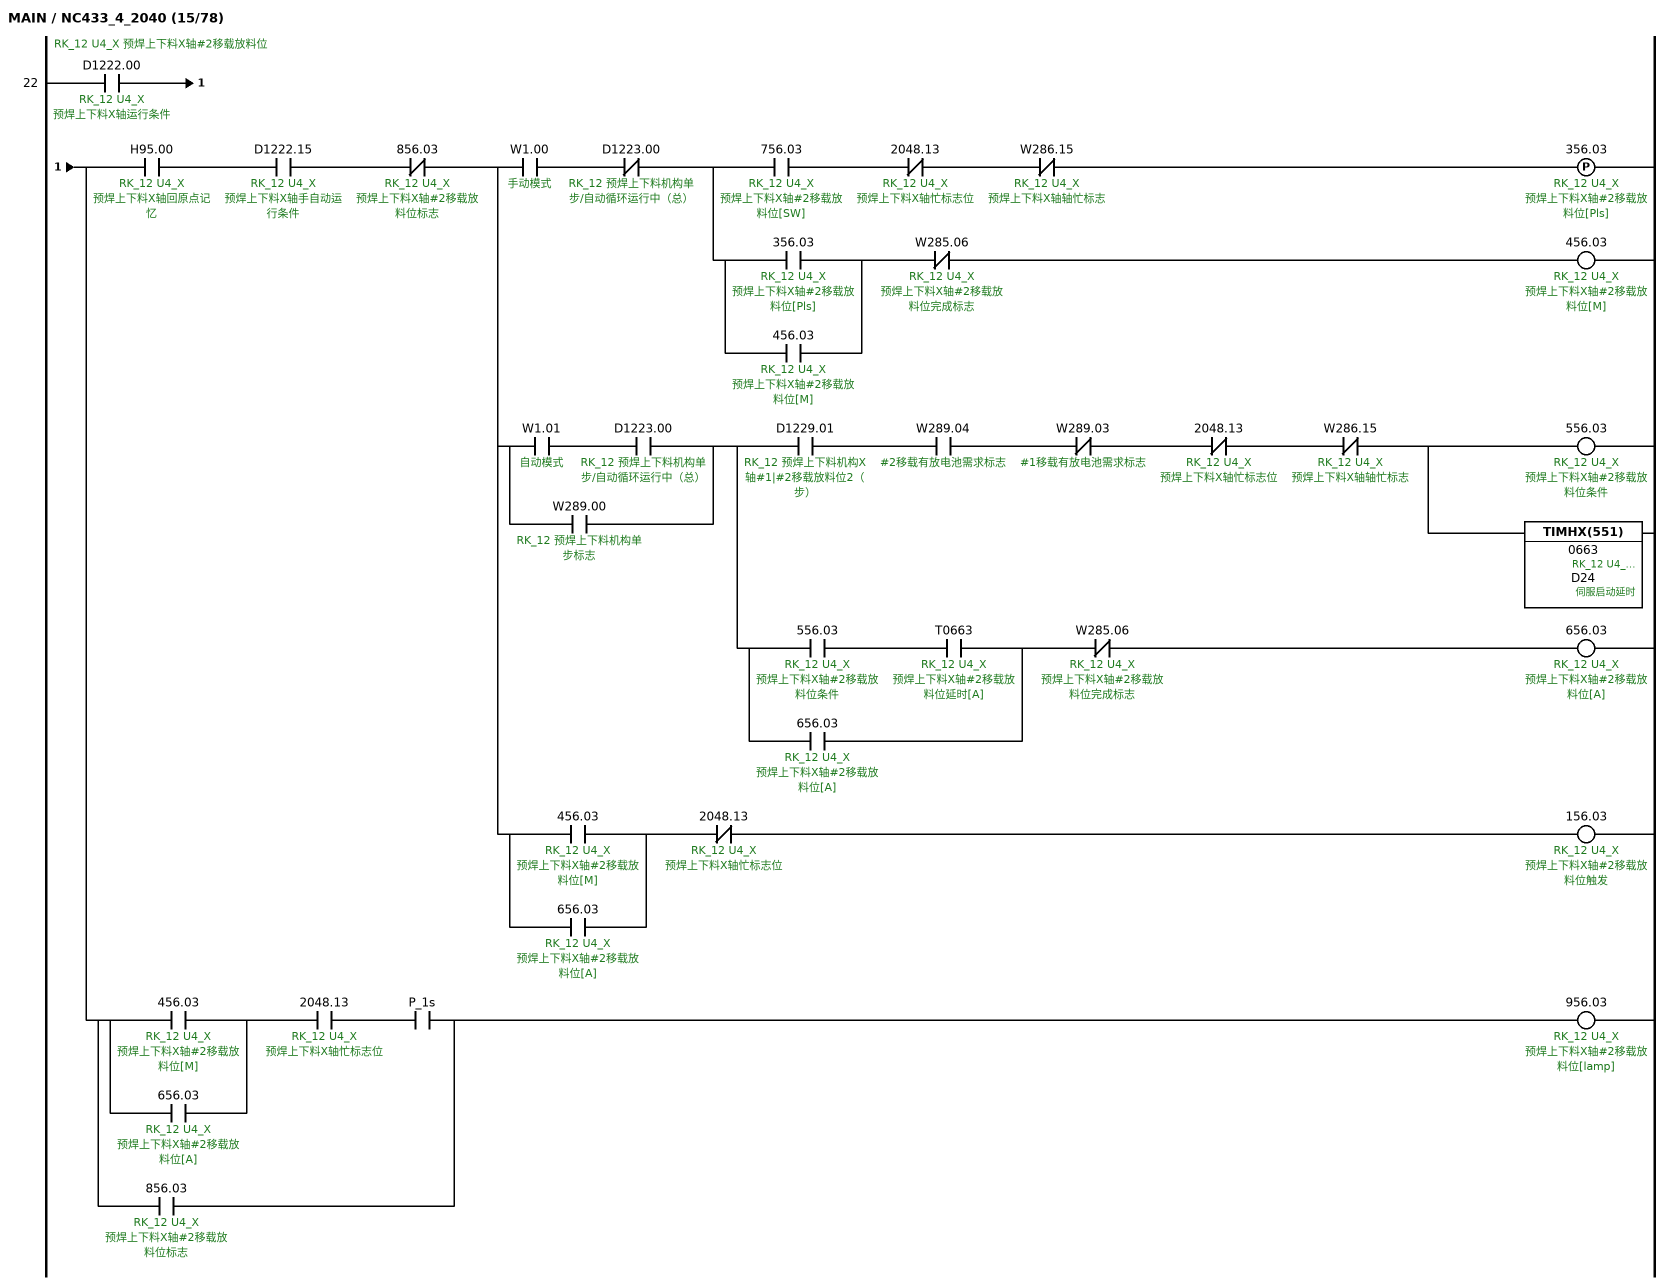
; rung 22: RK_12 U4_X 预焊上下料X轴#2移载放料位
LD D1222.00  ; RK_12 U4_X 预焊上下料X轴运行条件
OUT TR0
AND H95.00  ; RK_12 U4_X 预焊上下料X轴回原点记忆
AND D1222.15  ; RK_12 U4_X 预焊上下料X轴手自动运行条件
ANDNOT 856.03  ; RK_12 U4_X 预焊上下料X轴#2移载放料位标志
OUT TR1
AND W1.00  ; 手动模式
ANDNOT D1223.00  ; RK_12 预焊上下料机构单步/自动循环运行中（总）
OUT TR2
AND 756.03  ; RK_12 U4_X 预焊上下料X轴#2移载放料位[SW]
ANDNOT 2048.13  ; RK_12 U4_X 预焊上下料X轴忙标志位
ANDNOT W286.15  ; RK_12 U4_X 预焊上下料X轴轴忙标志
DIFU(013) 356.03  ; RK_12 U4_X 预焊上下料X轴#2移载放料位[Pls]
LD TR2
LD 356.03  ; RK_12 U4_X 预焊上下料X轴#2移载放料位[Pls]
OR 456.03  ; RK_12 U4_X 预焊上下料X轴#2移载放料位[M]
ANDLD
ANDNOT W285.06  ; RK_12 U4_X 预焊上下料X轴#2移载放料位完成标志
OUT 456.03  ; RK_12 U4_X 预焊上下料X轴#2移载放料位[M]
LD TR1
LD W1.01  ; 自动模式
AND D1223.00  ; RK_12 预焊上下料机构单步/自动循环运行中（总）
OR W289.00  ; RK_12 预焊上下料机构单步标志
ANDLD
OUT TR2
AND D1229.01  ; RK_12 预焊上下料机构X轴#1|#2移载放料位2（步）
AND W289.04  ; #2移载有放电池需求标志
ANDNOT W289.03  ; #1移载有放电池需求标志
ANDNOT 2048.13  ; RK_12 U4_X 预焊上下料X轴忙标志位
ANDNOT W286.15  ; RK_12 U4_X 预焊上下料X轴轴忙标志
OUT 556.03  ; RK_12 U4_X 预焊上下料X轴#2移载放料位条件
TIMHX(551) 0663 D24  ; 伺服启动延时, RK_12 U4_X 预焊上下料X轴#2移载放料位延时[A]
LD TR2
LD 556.03  ; RK_12 U4_X 预焊上下料X轴#2移载放料位条件
AND T0663  ; RK_12 U4_X 预焊上下料X轴#2移载放料位延时[A]
OR 656.03  ; RK_12 U4_X 预焊上下料X轴#2移载放料位[A]
ANDLD
ANDNOT W285.06  ; RK_12 U4_X 预焊上下料X轴#2移载放料位完成标志
OUT 656.03  ; RK_12 U4_X 预焊上下料X轴#2移载放料位[A]
LD TR1
LD 456.03  ; RK_12 U4_X 预焊上下料X轴#2移载放料位[M]
OR 656.03  ; RK_12 U4_X 预焊上下料X轴#2移载放料位[A]
ANDLD
ANDNOT 2048.13  ; RK_12 U4_X 预焊上下料X轴忙标志位
OUT 156.03  ; RK_12 U4_X 预焊上下料X轴#2移载放料位触发
LD TR0
LD 456.03  ; RK_12 U4_X 预焊上下料X轴#2移载放料位[M]
OR 656.03  ; RK_12 U4_X 预焊上下料X轴#2移载放料位[A]
AND 2048.13  ; RK_12 U4_X 预焊上下料X轴忙标志位
AND P_1s
OR 856.03  ; RK_12 U4_X 预焊上下料X轴#2移载放料位标志
ANDLD
OUT 956.03  ; RK_12 U4_X 预焊上下料X轴#2移载放料位[lamp]

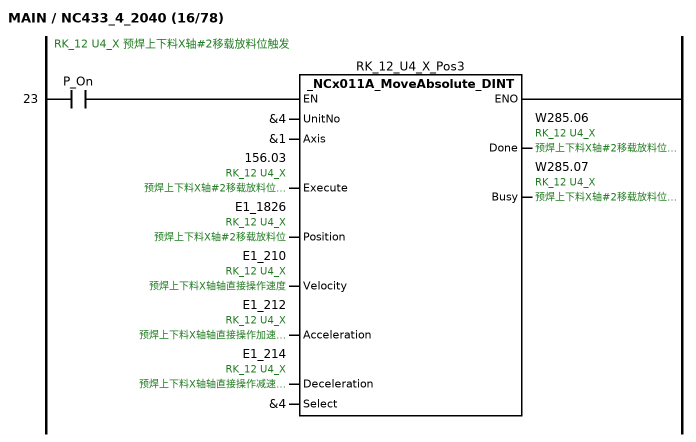
; rung 23: RK_12 U4_X 预焊上下料X轴#2移载放料位触发
LD P_On
CALL RK_12_U4_X_Pos3 : _NCx011A_MoveAbsolute_DINT (UnitNo := &4, Axis := &1, Execute := 156.03, Position := E1_1826, Velocity := E1_210, Acceleration := E1_212, Deceleration := E1_214, Select := &4, Done => W285.06, Busy => W285.07)  ; RK_12 U4_X 预焊上下料X轴#2移载放料位触发, RK_12 U4_X 预焊上下料X轴#2移载放料位, RK_12 U4_X 预焊上下料X轴轴直接操作速度, RK_12 U4_X 预焊上下料X轴轴直接操作加速时间, RK_12 U4_X 预焊上下料X轴轴直接操作减速时间, RK_12 U4_X 预焊上下料X轴#2移载放料位完成标志, RK_12 U4_X 预焊上下料X轴#2移载放料位忙标志

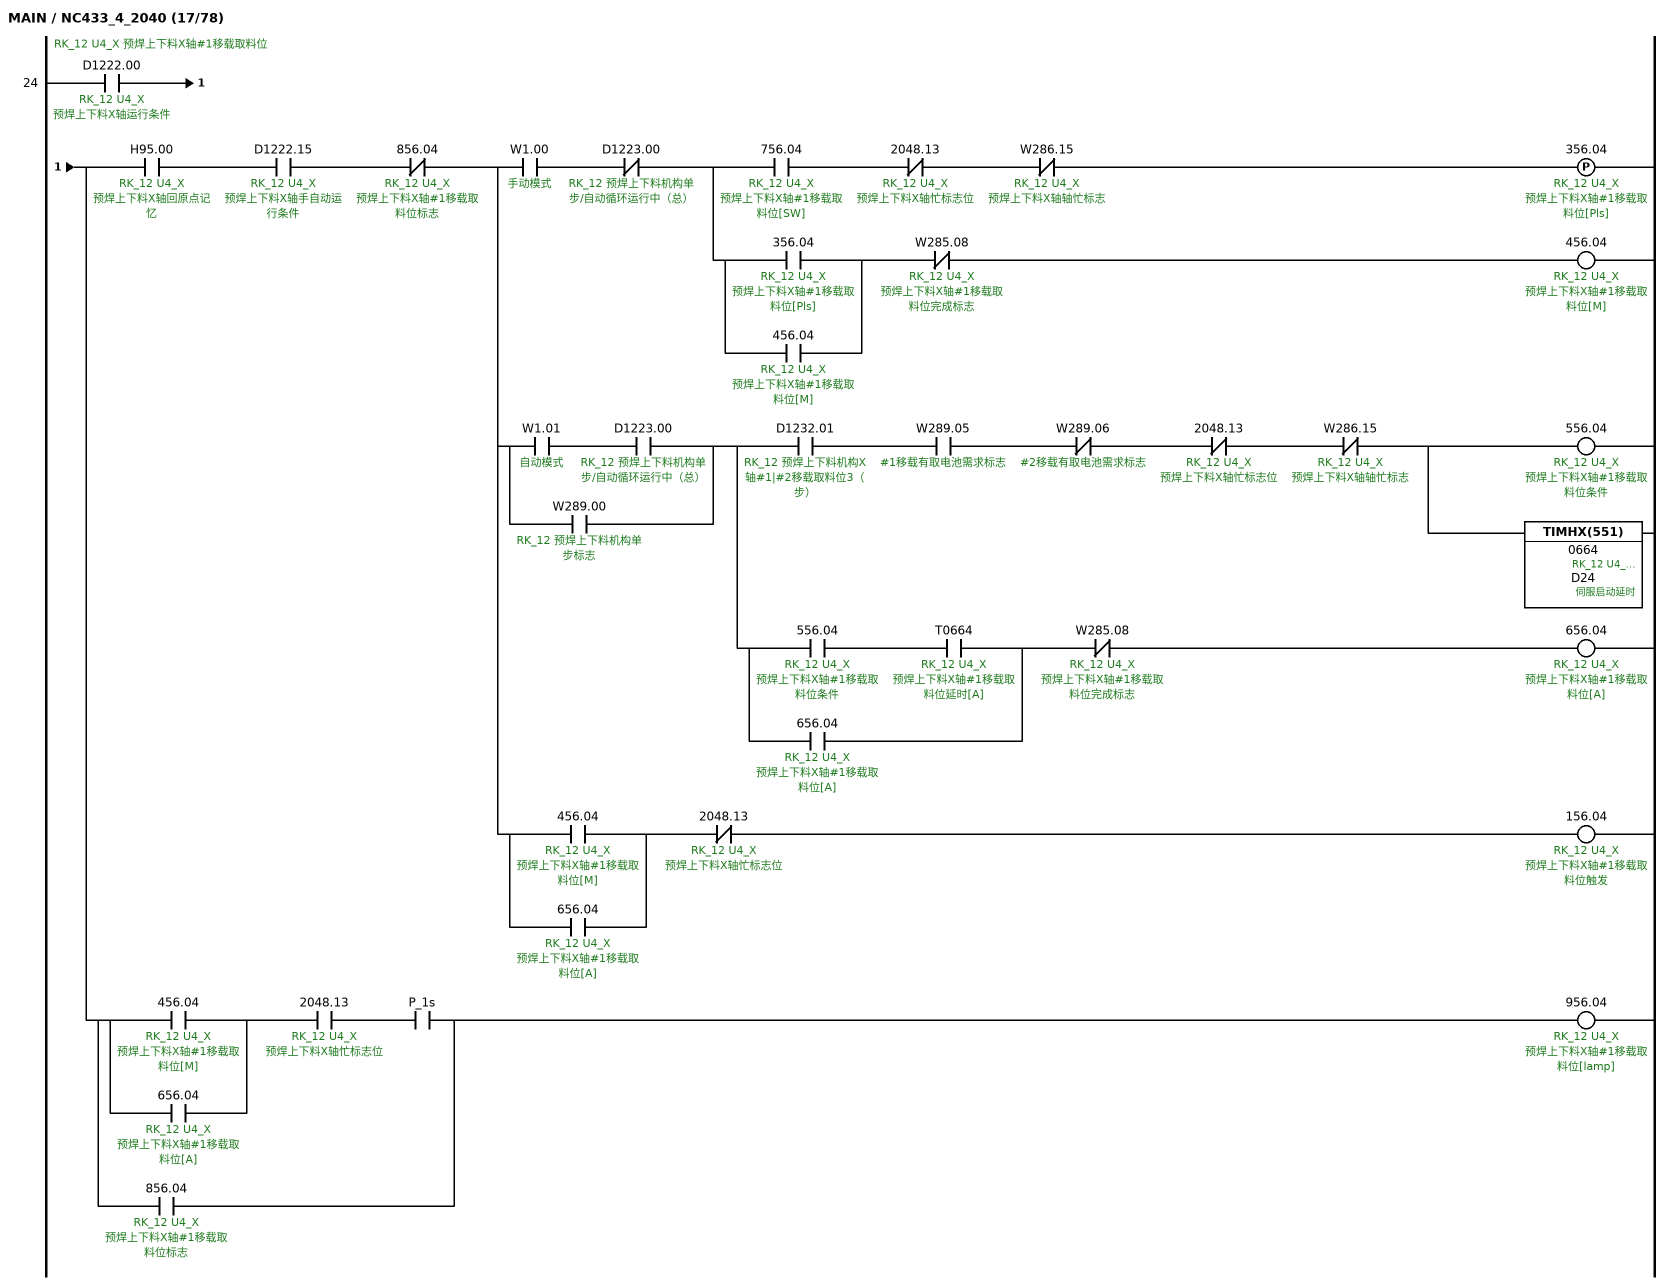
; rung 24: RK_12 U4_X 预焊上下料X轴#1移载取料位
LD D1222.00  ; RK_12 U4_X 预焊上下料X轴运行条件
OUT TR0
AND H95.00  ; RK_12 U4_X 预焊上下料X轴回原点记忆
AND D1222.15  ; RK_12 U4_X 预焊上下料X轴手自动运行条件
ANDNOT 856.04  ; RK_12 U4_X 预焊上下料X轴#1移载取料位标志
OUT TR1
AND W1.00  ; 手动模式
ANDNOT D1223.00  ; RK_12 预焊上下料机构单步/自动循环运行中（总）
OUT TR2
AND 756.04  ; RK_12 U4_X 预焊上下料X轴#1移载取料位[SW]
ANDNOT 2048.13  ; RK_12 U4_X 预焊上下料X轴忙标志位
ANDNOT W286.15  ; RK_12 U4_X 预焊上下料X轴轴忙标志
DIFU(013) 356.04  ; RK_12 U4_X 预焊上下料X轴#1移载取料位[Pls]
LD TR2
LD 356.04  ; RK_12 U4_X 预焊上下料X轴#1移载取料位[Pls]
OR 456.04  ; RK_12 U4_X 预焊上下料X轴#1移载取料位[M]
ANDLD
ANDNOT W285.08  ; RK_12 U4_X 预焊上下料X轴#1移载取料位完成标志
OUT 456.04  ; RK_12 U4_X 预焊上下料X轴#1移载取料位[M]
LD TR1
LD W1.01  ; 自动模式
AND D1223.00  ; RK_12 预焊上下料机构单步/自动循环运行中（总）
OR W289.00  ; RK_12 预焊上下料机构单步标志
ANDLD
OUT TR2
AND D1232.01  ; RK_12 预焊上下料机构X轴#1|#2移载取料位3（步）
AND W289.05  ; #1移载有取电池需求标志
ANDNOT W289.06  ; #2移载有取电池需求标志
ANDNOT 2048.13  ; RK_12 U4_X 预焊上下料X轴忙标志位
ANDNOT W286.15  ; RK_12 U4_X 预焊上下料X轴轴忙标志
OUT 556.04  ; RK_12 U4_X 预焊上下料X轴#1移载取料位条件
TIMHX(551) 0664 D24  ; 伺服启动延时, RK_12 U4_X 预焊上下料X轴#1移载取料位延时[A]
LD TR2
LD 556.04  ; RK_12 U4_X 预焊上下料X轴#1移载取料位条件
AND T0664  ; RK_12 U4_X 预焊上下料X轴#1移载取料位延时[A]
OR 656.04  ; RK_12 U4_X 预焊上下料X轴#1移载取料位[A]
ANDLD
ANDNOT W285.08  ; RK_12 U4_X 预焊上下料X轴#1移载取料位完成标志
OUT 656.04  ; RK_12 U4_X 预焊上下料X轴#1移载取料位[A]
LD TR1
LD 456.04  ; RK_12 U4_X 预焊上下料X轴#1移载取料位[M]
OR 656.04  ; RK_12 U4_X 预焊上下料X轴#1移载取料位[A]
ANDLD
ANDNOT 2048.13  ; RK_12 U4_X 预焊上下料X轴忙标志位
OUT 156.04  ; RK_12 U4_X 预焊上下料X轴#1移载取料位触发
LD TR0
LD 456.04  ; RK_12 U4_X 预焊上下料X轴#1移载取料位[M]
OR 656.04  ; RK_12 U4_X 预焊上下料X轴#1移载取料位[A]
AND 2048.13  ; RK_12 U4_X 预焊上下料X轴忙标志位
AND P_1s
OR 856.04  ; RK_12 U4_X 预焊上下料X轴#1移载取料位标志
ANDLD
OUT 956.04  ; RK_12 U4_X 预焊上下料X轴#1移载取料位[lamp]

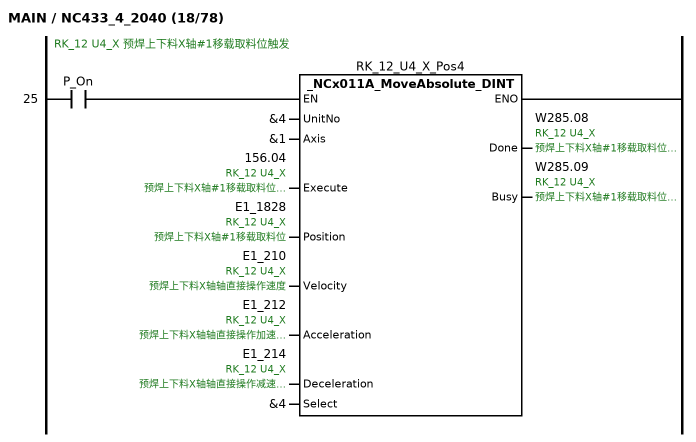
; rung 25: RK_12 U4_X 预焊上下料X轴#1移载取料位触发
LD P_On
CALL RK_12_U4_X_Pos4 : _NCx011A_MoveAbsolute_DINT (UnitNo := &4, Axis := &1, Execute := 156.04, Position := E1_1828, Velocity := E1_210, Acceleration := E1_212, Deceleration := E1_214, Select := &4, Done => W285.08, Busy => W285.09)  ; RK_12 U4_X 预焊上下料X轴#1移载取料位触发, RK_12 U4_X 预焊上下料X轴#1移载取料位, RK_12 U4_X 预焊上下料X轴轴直接操作速度, RK_12 U4_X 预焊上下料X轴轴直接操作加速时间, RK_12 U4_X 预焊上下料X轴轴直接操作减速时间, RK_12 U4_X 预焊上下料X轴#1移载取料位完成标志, RK_12 U4_X 预焊上下料X轴#1移载取料位忙标志

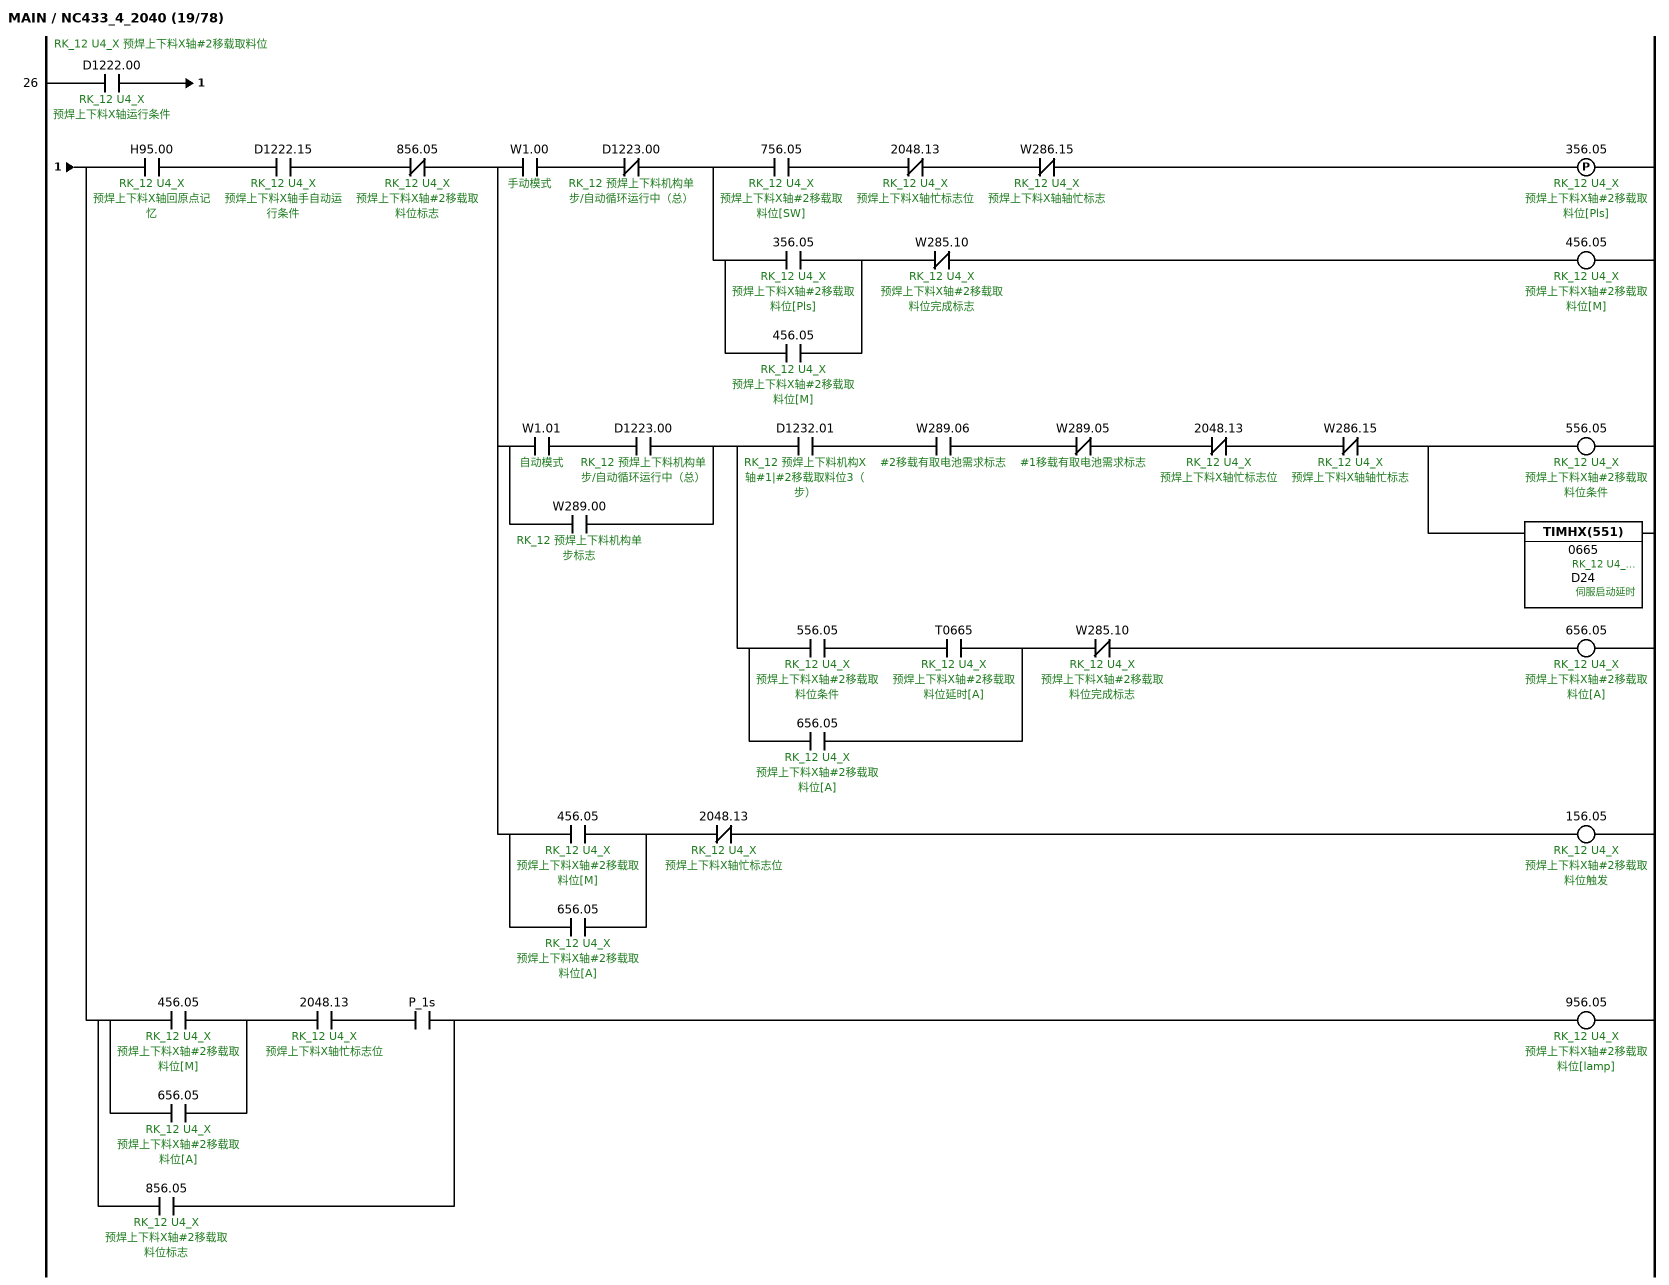
; rung 26: RK_12 U4_X 预焊上下料X轴#2移载取料位
LD D1222.00  ; RK_12 U4_X 预焊上下料X轴运行条件
OUT TR0
AND H95.00  ; RK_12 U4_X 预焊上下料X轴回原点记忆
AND D1222.15  ; RK_12 U4_X 预焊上下料X轴手自动运行条件
ANDNOT 856.05  ; RK_12 U4_X 预焊上下料X轴#2移载取料位标志
OUT TR1
AND W1.00  ; 手动模式
ANDNOT D1223.00  ; RK_12 预焊上下料机构单步/自动循环运行中（总）
OUT TR2
AND 756.05  ; RK_12 U4_X 预焊上下料X轴#2移载取料位[SW]
ANDNOT 2048.13  ; RK_12 U4_X 预焊上下料X轴忙标志位
ANDNOT W286.15  ; RK_12 U4_X 预焊上下料X轴轴忙标志
DIFU(013) 356.05  ; RK_12 U4_X 预焊上下料X轴#2移载取料位[Pls]
LD TR2
LD 356.05  ; RK_12 U4_X 预焊上下料X轴#2移载取料位[Pls]
OR 456.05  ; RK_12 U4_X 预焊上下料X轴#2移载取料位[M]
ANDLD
ANDNOT W285.10  ; RK_12 U4_X 预焊上下料X轴#2移载取料位完成标志
OUT 456.05  ; RK_12 U4_X 预焊上下料X轴#2移载取料位[M]
LD TR1
LD W1.01  ; 自动模式
AND D1223.00  ; RK_12 预焊上下料机构单步/自动循环运行中（总）
OR W289.00  ; RK_12 预焊上下料机构单步标志
ANDLD
OUT TR2
AND D1232.01  ; RK_12 预焊上下料机构X轴#1|#2移载取料位3（步）
AND W289.06  ; #2移载有取电池需求标志
ANDNOT W289.05  ; #1移载有取电池需求标志
ANDNOT 2048.13  ; RK_12 U4_X 预焊上下料X轴忙标志位
ANDNOT W286.15  ; RK_12 U4_X 预焊上下料X轴轴忙标志
OUT 556.05  ; RK_12 U4_X 预焊上下料X轴#2移载取料位条件
TIMHX(551) 0665 D24  ; 伺服启动延时, RK_12 U4_X 预焊上下料X轴#2移载取料位延时[A]
LD TR2
LD 556.05  ; RK_12 U4_X 预焊上下料X轴#2移载取料位条件
AND T0665  ; RK_12 U4_X 预焊上下料X轴#2移载取料位延时[A]
OR 656.05  ; RK_12 U4_X 预焊上下料X轴#2移载取料位[A]
ANDLD
ANDNOT W285.10  ; RK_12 U4_X 预焊上下料X轴#2移载取料位完成标志
OUT 656.05  ; RK_12 U4_X 预焊上下料X轴#2移载取料位[A]
LD TR1
LD 456.05  ; RK_12 U4_X 预焊上下料X轴#2移载取料位[M]
OR 656.05  ; RK_12 U4_X 预焊上下料X轴#2移载取料位[A]
ANDLD
ANDNOT 2048.13  ; RK_12 U4_X 预焊上下料X轴忙标志位
OUT 156.05  ; RK_12 U4_X 预焊上下料X轴#2移载取料位触发
LD TR0
LD 456.05  ; RK_12 U4_X 预焊上下料X轴#2移载取料位[M]
OR 656.05  ; RK_12 U4_X 预焊上下料X轴#2移载取料位[A]
AND 2048.13  ; RK_12 U4_X 预焊上下料X轴忙标志位
AND P_1s
OR 856.05  ; RK_12 U4_X 预焊上下料X轴#2移载取料位标志
ANDLD
OUT 956.05  ; RK_12 U4_X 预焊上下料X轴#2移载取料位[lamp]

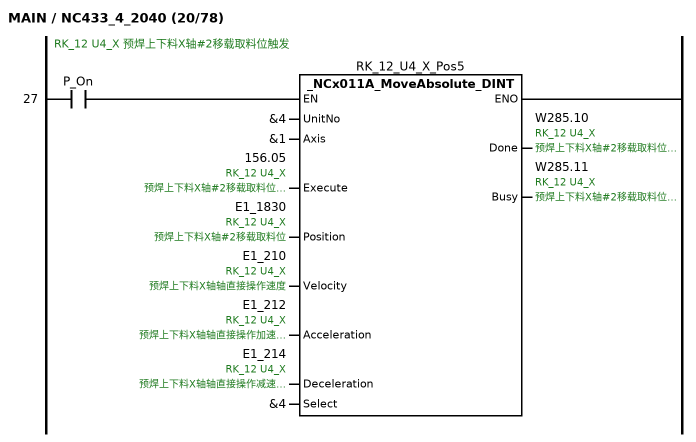
; rung 27: RK_12 U4_X 预焊上下料X轴#2移载取料位触发
LD P_On
CALL RK_12_U4_X_Pos5 : _NCx011A_MoveAbsolute_DINT (UnitNo := &4, Axis := &1, Execute := 156.05, Position := E1_1830, Velocity := E1_210, Acceleration := E1_212, Deceleration := E1_214, Select := &4, Done => W285.10, Busy => W285.11)  ; RK_12 U4_X 预焊上下料X轴#2移载取料位触发, RK_12 U4_X 预焊上下料X轴#2移载取料位, RK_12 U4_X 预焊上下料X轴轴直接操作速度, RK_12 U4_X 预焊上下料X轴轴直接操作加速时间, RK_12 U4_X 预焊上下料X轴轴直接操作减速时间, RK_12 U4_X 预焊上下料X轴#2移载取料位完成标志, RK_12 U4_X 预焊上下料X轴#2移载取料位忙标志

